SPLINE
SPL {X  -159.701, Y  +348.785, Z    +0.000, E1   +24.361, E3 +434881.176}
SPL {X  -161.904, Y  +363.251, Z    +0.000, E1   +14.606, E3 +434910.971}
SPL {X  -162.745, Y  +375.561, Z    +0.000, E1    +7.538, E3 +434911.168}
SPL {X  -162.820, Y  +385.424, Z    +0.000, E1    +1.080, E3 +434912.062}
SPL {X  -162.820, Y  +389.940, Z    +0.000, E1    -2.281, E3 +434914.938}
SPL {X  -162.820, Y  +396.652, Z    +0.000, E1    -7.520, E3 +434914.517}
SPL {X  -162.820, Y  +406.605, Z    +0.000, E1   -16.760, E3 +434906.994}
SPL {X  -162.820, Y  +420.013, Z    +0.000, E1   -22.833, E3 +434935.115}
SPL {X  -162.820, Y  +442.075, Z    +0.000, E1   -31.090, E3 +434967.901}
ENDSPLINE

SPLINE
SPL {X  -162.820, Y  +436.680, Z    +0.000, E1   -26.151, E3 +434981.205}
ENDSPLINE

SPLINE
SPL {X  -162.820, Y  +438.487, Z    +0.000, E1   -25.409, E3 +434994.844}
SPL {X  -162.820, Y  +441.593, Z    +0.000, E1   -25.391, E3 +435008.452}
SPL {X  -162.820, Y  +444.317, Z    +0.000, E1   -25.492, E3 +435019.634}
SPL {X  -162.820, Y  +446.544, Z    +0.000, E1   -25.427, E3 +435029.803}
SPL {X  -162.820, Y  +448.500, Z    +0.000, E1   -25.425, E3 +435038.405}
SPL {X  -162.820, Y  +451.056, Z    +0.000, E1   -25.443, E3 +435049.512}
SPL {X  -162.820, Y  +454.662, Z    +0.000, E1   -25.474, E3 +435065.256}
SPL {X  -162.820, Y  +458.079, Z    +0.000, E1   -25.369, E3 +435080.835}
SPL {X  -162.820, Y  +460.719, Z    +0.000, E1   -25.411, E3 +435092.094}
SPL {X  -162.820, Y  +463.419, Z    +0.000, E1   -25.510, E3 +435103.131}
SPL {X  -162.820, Y  +465.376, Z    +0.000, E1   -25.372, E3 +435112.719}
SPL {X  -162.820, Y  +467.440, Z    +0.000, E1   -25.427, E3 +435121.351}
SPL {X  -162.820, Y  +470.010, Z    +0.000, E1   -25.445, E3 +435132.555}
SPL {X  -162.820, Y  +473.445, Z    +0.000, E1   -25.493, E3 +435147.279}
SPL {X  -162.820, Y  +476.157, Z    +0.000, E1   -25.426, E3 +435159.494}
SPL {X  -162.820, Y  +478.461, Z    +0.000, E1   -25.410, E3 +435169.774}
SPL {X  -162.820, Y  +481.644, Z    +0.000, E1   -25.433, E3 +435183.720}
SPL {X  -162.820, Y  +486.042, Z    +0.000, E1   -25.483, E3 +435202.639}
SPL {X  -162.820, Y  +490.287, Z    +0.000, E1   -25.463, E3 +435221.358}
SPL {X  -162.820, Y  +494.454, Z    +0.000, E1   -25.465, E3 +435239.589}
SPL {X  -162.820, Y  +498.644, Z    +0.000, E1   -25.463, E3 +435257.965}
SPL {X  -162.820, Y  +502.845, Z    +0.000, E1   -25.458, E3 +435276.399}
SPL {X  -162.820, Y  +506.050, Z    +0.000, E1   -25.420, E3 +435290.538}
SPL {X  -162.820, Y  +508.346, Z    +0.000, E1   -25.444, E3 +435300.387}
SPL {X  -162.820, Y  +511.422, Z    +0.000, E1   -25.445, E3 +435314.047}
SPL {X  -162.820, Y  +515.039, Z    +0.000, E1   -25.452, E3 +435329.728}
SPL {X  -162.820, Y  +517.481, Z    +0.000, E1   -25.432, E3 +435340.463}
SPL {X  -162.820, Y  +519.134, Z    +0.000, E1   -25.366, E3 +435348.210}
SPL {X  -162.820, Y  +521.486, Z    +0.000, E1   -25.382, E3 +435358.506}
SPL {X  -162.820, Y  +525.073, Z    +0.000, E1   -25.512, E3 +435373.312}
SPL {X  -162.820, Y  +527.738, Z    +0.000, E1   -25.438, E3 +435385.360}
SPL {X  -162.820, Y  +530.432, Z    +0.000, E1   -25.477, E3 +435396.937}
SPL {X  -162.820, Y  +534.051, Z    +0.000, E1   -25.484, E3 +435412.814}
SPL {X  -162.820, Y  +537.226, Z    +0.000, E1   -25.378, E3 +435427.383}
SPL {X  -162.820, Y  +539.521, Z    +0.000, E1   -25.386, E3 +435437.342}
SPL {X  -162.820, Y  +542.667, Z    +0.000, E1   -25.474, E3 +435450.667}
SPL {X  -162.820, Y  +546.125, Z    +0.000, E1   -25.505, E3 +435465.392}
SPL {X  -162.820, Y  +548.232, Z    +0.000, E1   -25.424, E3 +435475.154}
SPL {X  -162.820, Y  +550.399, Z    +0.000, E1   -25.424, E3 +435484.705}
SPL {X  -162.820, Y  +553.157, Z    +0.000, E1   -25.443, E3 +435496.679}
SPL {X  -162.820, Y  +556.150, Z    +0.000, E1   -25.445, E3 +435509.769}
SPL {X  -162.820, Y  +559.215, Z    +0.000, E1   -25.460, E3 +435523.071}
SPL {X  -162.820, Y  +562.125, Z    +0.000, E1   -25.434, E3 +435535.991}
SPL {X  -162.820, Y  +564.880, Z    +0.000, E1   -25.448, E3 +435547.945}
SPL {X  -162.820, Y  +568.326, Z    +0.000, E1   -25.470, E3 +435563.005}
SPL {X  -162.820, Y  +572.331, Z    +0.000, E1   -25.489, E3 +435580.380}
SPL {X  -162.820, Y  +576.045, Z    +0.000, E1   -25.412, E3 +435597.188}
SPL {X  -162.820, Y  +580.038, Z    +0.000, E1   -25.473, E3 +435614.283}
SPL {X  -162.820, Y  +583.044, Z    +0.000, E1   -25.450, E3 +435627.406}
SPL {X  -162.820, Y  +585.512, Z    +0.000, E1   -25.448, E3 +435638.302}
SPL {X  -162.820, Y  +588.371, Z    +0.000, E1   -25.460, E3 +435650.688}
SPL {X  -162.820, Y  +590.476, Z    +0.000, E1   -25.398, E3 +435660.329}
SPL {X  -162.820, Y  +593.604, Z    +0.000, E1   -25.477, E3 +435673.607}
SPL {X  -162.820, Y  +596.868, Z    +0.000, E1   -25.461, E3 +435687.873}
SPL {X  -162.820, Y  +599.135, Z    +0.000, E1   -25.398, E3 +435698.242}
SPL {X  -162.820, Y  +601.296, Z    +0.000, E1   -25.399, E3 +435707.723}
SPL {X  -162.820, Y  +603.808, Z    +0.000, E1   -25.554, E3 +435717.511}
SPL {X  -162.820, Y  +607.007, Z    +0.000, E1   -25.491, E3 +435732.202}
SPL {X  -162.820, Y  +611.438, Z    +0.000, E1   -25.467, E3 +435751.792}
SPL {X  -162.820, Y  +615.388, Z    +0.000, E1   -25.455, E3 +435769.051}
SPL {X  -162.820, Y  +618.995, Z    +0.000, E1   -25.483, E3 +435784.646}
SPL {X  -162.820, Y  +622.118, Z    +0.000, E1   -25.492, E3 +435798.111}
SPL {X  -162.820, Y  +624.430, Z    +0.000, E1   -25.475, E3 +435808.332}
SPL {X  -162.820, Y  +626.570, Z    +0.000, E1   -25.441, E3 +435817.932}
SPL {X  -162.820, Y  +628.902, Z    +0.000, E1   -25.449, E3 +435828.113}
SPL {X  -162.820, Y  +631.177, Z    +0.000, E1   -25.467, E3 +435837.944}
SPL {X  -162.820, Y  +633.994, Z    +0.000, E1   -25.503, E3 +435849.990}
SPL {X  -162.820, Y  +636.469, Z    +0.000, E1   -25.465, E3 +435861.034}
SPL {X  -162.820, Y  +638.486, Z    +0.000, E1   -25.456, E3 +435869.952}
SPL {X  -162.820, Y  +640.803, Z    +0.000, E1   -25.462, E3 +435880.013}
SPL {X  -162.820, Y  +643.028, Z    +0.000, E1   -25.494, E3 +435889.522}
SPL {X  -162.820, Y  +645.694, Z    +0.000, E1   -25.540, E3 +435900.810}
SPL {X  -162.820, Y  +649.102, Z    +0.000, E1   -25.495, E3 +435916.238}
SPL {X  -162.820, Y  +652.810, Z    +0.000, E1   -25.497, E3 +435932.272}
SPL {X  -162.820, Y  +655.214, Z    +0.000, E1   -25.485, E3 +435942.774}
SPL {X  -162.820, Y  +657.616, Z    +0.000, E1   -25.511, E3 +435953.129}
SPL {X  -162.820, Y  +660.851, Z    +0.000, E1   -25.520, E3 +435967.271}
SPL {X  -162.820, Y  +663.853, Z    +0.000, E1   -25.496, E3 +435980.453}
SPL {X  -162.820, Y  +667.253, Z    +0.000, E1   -25.483, E3 +435995.625}
SPL {X  -162.820, Y  +671.102, Z    +0.000, E1   -25.514, E3 +436012.076}
SPL {X  -162.820, Y  +673.648, Z    +0.000, E1   -25.431, E3 +436023.742}
SPL {X  -162.796, Y  +676.319, Z    +0.000, E1   -25.526, E3 +436034.752}
SPL {X  -162.707, Y  +679.552, Z    +0.000, E1   -25.443, E3 +436049.626}
SPL {X  -162.545, Y  +682.952, Z    +0.000, E1   -25.510, E3 +436063.859}
SPL {X  -162.381, Y  +685.455, Z    +0.000, E1   -25.410, E3 +436075.546}
SPL {X  -162.194, Y  +687.760, Z    +0.000, E1   -25.360, E3 +436085.982}
SPL {X  -161.866, Y  +691.104, Z    +0.000, E1   -25.383, E3 +436100.614}
SPL {X  -161.319, Y  +695.558, Z    +0.000, E1   -25.832, E3 +436116.416}
SPL {X  -157.976, Y  +712.921, Z    +0.000, E1   -33.197, E3 +436129.808}
ENDSPLINE

SPLINE
SPL {X  -160.738, Y  +699.453, Z    +0.000, E1   -21.994, E3 +436167.435}
SPL {X  -160.945, Y  +698.140, Z    +0.000, E1   -18.412, E3 +436209.674}
SPL {X  -162.497, Y  +683.755, Z    +0.000, E1   -10.754, E3 +436203.818}
SPL {X  -162.819, Y  +673.996, Z    +0.000, E1    -4.745, E3 +436203.419}
ENDSPLINE

SPLINE
SPL {X  -162.791, Y  +676.574, Z    +0.000, E1    -6.127, E3 +436216.107}
ENDSPLINE

SPLINE
SPL {X  -162.820, Y  +667.935, Z    +0.000, E1    -0.509, E3 +436206.193}
SPL {X  -162.820, Y  +662.949, Z    +0.000, E1    +3.113, E3 +436204.312}
SPL {X  -162.820, Y  +658.484, Z    +0.000, E1    +6.336, E3 +436211.457}
SPL {X  -162.820, Y  +640.102, Z    +0.000, E1   +22.409, E3 +436206.196}
SPL {X  -162.820, Y  +633.503, Z    +0.000, E1   +21.975, E3 +436238.433}
SPL {X  -162.820, Y  +611.299, Z    +0.000, E1   +31.088, E3 +436266.545}
ENDSPLINE

SPLINE
SPL {X  -162.820, Y  +618.877, Z    +0.000, E1   +25.259, E3 +436278.040}
ENDSPLINE

SPLINE
SPL {X  -162.820, Y  +617.582, Z    +0.000, E1   +24.552, E3 +436289.416}
SPL {X  -162.820, Y  +614.716, Z    +0.000, E1   +24.535, E3 +436302.628}
SPL {X  -162.820, Y  +611.754, Z    +0.000, E1   +24.563, E3 +436315.916}
SPL {X  -162.820, Y  +608.970, Z    +0.000, E1   +24.542, E3 +436328.756}
SPL {X  -162.820, Y  +606.285, Z    +0.000, E1   +24.533, E3 +436341.092}
SPL {X  -162.820, Y  +603.509, Z    +0.000, E1   +24.546, E3 +436353.629}
SPL {X  -162.820, Y  +600.230, Z    +0.000, E1   +24.589, E3 +436368.374}
SPL {X  -162.820, Y  +597.446, Z    +0.000, E1   +24.542, E3 +436381.232}
SPL {X  -162.820, Y  +595.188, Z    +0.000, E1   +24.538, E3 +436391.623}
SPL {X  -162.820, Y  +592.738, Z    +0.000, E1   +24.551, E3 +436402.671}
SPL {X  -162.820, Y  +590.118, Z    +0.000, E1   +24.544, E3 +436414.731}
SPL {X  -162.820, Y  +587.204, Z    +0.000, E1   +24.592, E3 +436427.607}
SPL {X  -162.820, Y  +584.766, Z    +0.000, E1   +24.499, E3 +436439.441}
SPL {X  -162.820, Y  +581.896, Z    +0.000, E1   +24.528, E3 +436452.383}
SPL {X  -162.820, Y  +579.244, Z    +0.000, E1   +24.610, E3 +436463.727}
SPL {X  -162.820, Y  +576.848, Z    +0.000, E1   +24.543, E3 +436475.268}
SPL {X  -162.820, Y  +573.694, Z    +0.000, E1   +24.535, E3 +436489.738}
SPL {X  -162.820, Y  +571.322, Z    +0.000, E1   +24.492, E3 +436500.771}
SPL {X  -162.820, Y  +568.309, Z    +0.000, E1   +24.589, E3 +436513.996}
SPL {X  -162.820, Y  +564.977, Z    +0.000, E1   +24.571, E3 +436529.169}
SPL {X  -162.820, Y  +562.356, Z    +0.000, E1   +24.575, E3 +436541.068}
SPL {X  -162.820, Y  +558.990, Z    +0.000, E1   +24.558, E3 +436556.718}
SPL {X  -162.820, Y  +555.584, Z    +0.000, E1   +24.559, E3 +436572.087}
SPL {X  -162.820, Y  +552.867, Z    +0.000, E1   +24.583, E3 +436584.282}
SPL {X  -162.820, Y  +549.589, Z    +0.000, E1   +24.547, E3 +436599.648}
SPL {X  -162.820, Y  +546.972, Z    +0.000, E1   +24.516, E3 +436611.613}
SPL {X  -162.820, Y  +544.025, Z    +0.000, E1   +24.611, E3 +436624.558}
SPL {X  -162.820, Y  +540.573, Z    +0.000, E1   +24.503, E3 +436641.012}
SPL {X  -162.820, Y  +538.106, Z    +0.000, E1   +24.553, E3 +436651.766}
SPL {X  -162.820, Y  +536.451, Z    +0.000, E1   +24.519, E3 +436659.584}
SPL {X  -162.820, Y  +534.025, Z    +0.000, E1   +24.589, E3 +436670.184}
SPL {X  -162.820, Y  +531.527, Z    +0.000, E1   +24.582, E3 +436681.570}
SPL {X  -162.820, Y  +529.165, Z    +0.000, E1   +24.521, E3 +436692.819}
SPL {X  -162.820, Y  +525.802, Z    +0.000, E1   +24.585, E3 +436707.839}
SPL {X  -162.820, Y  +521.731, Z    +0.000, E1   +24.542, E3 +436726.775}
SPL {X  -162.820, Y  +518.185, Z    +0.000, E1   +24.561, E3 +436742.647}
SPL {X  -162.820, Y  +508.728, Z    +0.000, E1   +28.484, E3 +436753.187}
SPL {X  -162.820, Y  +500.664, Z    +0.000, E1   +31.476, E3 +436761.851}
SPL {X  -162.820, Y  +499.290, Z    +0.000, E1   +30.657, E3 +436772.133}
SPL {X  -162.820, Y  +497.251, Z    +0.000, E1   +29.634, E3 +436786.608}
SPL {X  -162.820, Y  +495.647, Z    +0.000, E1   +28.606, E3 +436799.485}
SPL {X  -162.820, Y  +494.678, Z    +0.000, E1   +27.647, E3 +436810.186}
SPL {X  -162.820, Y  +493.757, Z    +0.000, E1   +26.462, E3 +436822.546}
SPL {X  -162.820, Y  +492.330, Z    +0.000, E1   +25.953, E3 +436832.300}
SPL {X  -162.820, Y  +489.800, Z    +0.000, E1   +25.653, E3 +436845.761}
SPL {X  -162.820, Y  +485.392, Z    +0.000, E1   +25.667, E3 +436864.789}
SPL {X  -162.820, Y  +482.092, Z    +0.000, E1   +25.593, E3 +436879.477}
SPL {X  -162.820, Y  +479.578, Z    +0.000, E1   +25.634, E3 +436890.120}
SPL {X  -162.820, Y  +477.137, Z    +0.000, E1   +25.632, E3 +436900.699}
SPL {X  -162.820, Y  +473.770, Z    +0.000, E1   +25.664, E3 +436915.245}
SPL {X  -162.820, Y  +469.694, Z    +0.000, E1   +25.657, E3 +436932.976}
SPL {X  -162.820, Y  +465.727, Z    +0.000, E1   +25.676, E3 +436950.019}
SPL {X  -162.820, Y  +463.001, Z    +0.000, E1   +25.614, E3 +436962.135}
SPL {X  -162.820, Y  +459.882, Z    +0.000, E1   +25.674, E3 +436975.435}
SPL {X  -162.820, Y  +456.773, Z    +0.000, E1   +25.591, E3 +436989.382}
SPL {X  -162.820, Y  +454.429, Z    +0.000, E1   +25.642, E3 +436999.149}
SPL {X  -162.820, Y  +451.204, Z    +0.000, E1   +25.672, E3 +437013.176}
SPL {X  -162.820, Y  +447.822, Z    +0.000, E1   +25.664, E3 +437027.660}
SPL {X  -162.820, Y  +445.556, Z    +0.000, E1   +25.626, E3 +437037.791}
SPL {X  -162.820, Y  +442.508, Z    +0.000, E1   +25.657, E3 +437050.885}
SPL {X  -162.820, Y  +439.273, Z    +0.000, E1   +25.576, E3 +437065.522}
SPL {X  -162.820, Y  +436.773, Z    +0.000, E1   +25.602, E3 +437076.087}
SPL {X  -162.820, Y  +433.761, Z    +0.000, E1   +25.681, E3 +437088.766}
SPL {X  -162.820, Y  +430.942, Z    +0.000, E1   +25.597, E3 +437101.451}
SPL {X  -162.820, Y  +428.576, Z    +0.000, E1   +25.647, E3 +437111.389}
SPL {X  -162.820, Y  +426.525, Z    +0.000, E1   +25.610, E3 +437120.496}
SPL {X  -162.820, Y  +423.655, Z    +0.000, E1   +25.628, E3 +437133.056}
SPL {X  -162.820, Y  +419.407, Z    +0.000, E1   +25.665, E3 +437151.248}
SPL {X  -162.820, Y  +415.900, Z    +0.000, E1   +25.638, E3 +437166.517}
SPL {X  -162.820, Y  +413.088, Z    +0.000, E1   +25.644, E3 +437178.674}
SPL {X  -162.820, Y  +410.320, Z    +0.000, E1   +25.604, E3 +437190.992}
SPL {X  -162.820, Y  +407.487, Z    +0.000, E1   +25.617, E3 +437203.200}
SPL {X  -162.820, Y  +405.108, Z    +0.000, E1   +25.535, E3 +437214.168}
SPL {X  -162.820, Y  +401.373, Z    +0.000, E1   +25.736, E3 +437229.004}
SPL {X  -162.820, Y  +398.703, Z    +0.000, E1   +25.586, E3 +437241.501}
SPL {X  -162.820, Y  +395.582, Z    +0.000, E1   +25.684, E3 +437254.493}
SPL {X  -162.820, Y  +391.417, Z    +0.000, E1   +25.659, E3 +437272.831}
SPL {X  -162.820, Y  +387.939, Z    +0.000, E1   +25.627, E3 +437287.978}
SPL {X  -162.820, Y  +385.565, Z    +0.000, E1   +25.686, E3 +437297.766}
SPL {X  -162.820, Y  +383.458, Z    +0.000, E1   +25.657, E3 +437307.130}
SPL {X  -162.820, Y  +381.229, Z    +0.000, E1   +25.660, E3 +437316.806}
SPL {X  -162.797, Y  +377.786, Z    +0.000, E1   +25.638, E3 +437332.095}
SPL {X  -162.663, Y  +373.346, Z    +0.000, E1   +25.707, E3 +437350.834}
SPL {X  -162.487, Y  +370.088, Z    +0.000, E1   +25.525, E3 +437366.169}
SPL {X  -162.307, Y  +367.587, Z    +0.000, E1   +25.577, E3 +437376.587}
SPL {X  -162.041, Y  +364.588, Z    +0.000, E1   +25.591, E3 +437389.665}
SPL {X  -161.695, Y  +361.389, Z    +0.000, E1   +25.445, E3 +437404.551}
SPL {X  -161.190, Y  +357.520, Z    +0.000, E1   +25.774, E3 +437418.802}
SPL {X  -154.424, Y  +328.890, Z    +0.000, E1   +36.591, E3 +437443.802}
ENDSPLINE

SPLINE
SPL {X  -159.701, Y  +348.785, Z    +0.000, E1   +24.361, E3 +437472.085}
SPL {X  -161.904, Y  +363.251, Z    +0.000, E1   +14.606, E3 +437501.880}
SPL {X  -162.745, Y  +375.561, Z    +0.000, E1    +7.538, E3 +437502.077}
SPL {X  -162.820, Y  +385.424, Z    +0.000, E1    +1.080, E3 +437502.971}
SPL {X  -162.820, Y  +389.940, Z    +0.000, E1    -2.281, E3 +437505.847}
SPL {X  -162.820, Y  +396.652, Z    +0.000, E1    -7.520, E3 +437505.426}
SPL {X  -162.820, Y  +406.605, Z    +0.000, E1   -16.760, E3 +437497.903}
SPL {X  -162.820, Y  +418.675, Z    +0.000, E1   -22.201, E3 +437524.151}
SPL {X  -162.820, Y  +425.113, Z    +0.000, E1   -25.243, E3 +437533.088}
SPL {X  -162.820, Y  +442.075, Z    +0.000, E1   -31.090, E3 +437558.810}
ENDSPLINE

SPLINE
SPL {X  -162.820, Y  +436.949, Z    +0.000, E1   -25.871, E3 +437575.560}
ENDSPLINE

SPLINE
SPL {X  -162.820, Y  +439.120, Z    +0.000, E1   -25.352, E3 +437588.809}
SPL {X  -162.820, Y  +441.593, Z    +0.000, E1   -25.391, E3 +437599.361}
SPL {X  -162.820, Y  +444.317, Z    +0.000, E1   -25.492, E3 +437610.543}
SPL {X  -162.820, Y  +447.641, Z    +0.000, E1   -25.460, E3 +437625.478}
SPL {X  -162.820, Y  +451.056, Z    +0.000, E1   -25.443, E3 +437640.421}
SPL {X  -162.820, Y  +454.662, Z    +0.000, E1   -25.474, E3 +437656.165}
SPL {X  -162.820, Y  +458.079, Z    +0.000, E1   -25.369, E3 +437671.745}
SPL {X  -162.820, Y  +460.719, Z    +0.000, E1   -25.411, E3 +437683.003}
SPL {X  -162.820, Y  +463.419, Z    +0.000, E1   -25.510, E3 +437694.040}
SPL {X  -162.820, Y  +465.376, Z    +0.000, E1   -25.372, E3 +437703.628}
SPL {X  -162.820, Y  +467.440, Z    +0.000, E1   -25.427, E3 +437712.260}
SPL {X  -162.820, Y  +470.010, Z    +0.000, E1   -25.445, E3 +437723.464}
SPL {X  -162.820, Y  +473.445, Z    +0.000, E1   -25.493, E3 +437738.188}
SPL {X  -162.820, Y  +476.157, Z    +0.000, E1   -25.426, E3 +437750.403}
SPL {X  -162.820, Y  +478.461, Z    +0.000, E1   -25.410, E3 +437760.683}
SPL {X  -162.820, Y  +481.644, Z    +0.000, E1   -25.433, E3 +437774.629}
SPL {X  -162.820, Y  +486.042, Z    +0.000, E1   -25.483, E3 +437793.548}
SPL {X  -162.820, Y  +490.287, Z    +0.000, E1   -25.463, E3 +437812.267}
SPL {X  -162.820, Y  +494.454, Z    +0.000, E1   -25.465, E3 +437830.498}
SPL {X  -162.820, Y  +498.644, Z    +0.000, E1   -25.463, E3 +437848.874}
SPL {X  -162.820, Y  +502.845, Z    +0.000, E1   -25.458, E3 +437867.308}
SPL {X  -162.820, Y  +506.050, Z    +0.000, E1   -25.420, E3 +437881.447}
SPL {X  -162.820, Y  +508.346, Z    +0.000, E1   -25.444, E3 +437891.296}
SPL {X  -162.820, Y  +511.422, Z    +0.000, E1   -25.445, E3 +437904.956}
SPL {X  -162.820, Y  +515.039, Z    +0.000, E1   -25.452, E3 +437920.638}
SPL {X  -162.820, Y  +517.481, Z    +0.000, E1   -25.432, E3 +437931.372}
SPL {X  -162.820, Y  +519.134, Z    +0.000, E1   -25.366, E3 +437939.119}
SPL {X  -162.820, Y  +521.486, Z    +0.000, E1   -25.382, E3 +437949.415}
SPL {X  -162.820, Y  +525.073, Z    +0.000, E1   -25.512, E3 +437964.221}
SPL {X  -162.820, Y  +527.738, Z    +0.000, E1   -25.438, E3 +437976.269}
SPL {X  -162.820, Y  +530.432, Z    +0.000, E1   -25.477, E3 +437987.846}
SPL {X  -162.820, Y  +534.051, Z    +0.000, E1   -25.484, E3 +438003.723}
SPL {X  -162.820, Y  +537.226, Z    +0.000, E1   -25.378, E3 +438018.292}
SPL {X  -162.820, Y  +539.521, Z    +0.000, E1   -25.386, E3 +438028.251}
SPL {X  -162.820, Y  +542.667, Z    +0.000, E1   -25.474, E3 +438041.576}
SPL {X  -162.820, Y  +546.125, Z    +0.000, E1   -25.505, E3 +438056.301}
SPL {X  -162.820, Y  +549.578, Z    +0.000, E1   -25.462, E3 +438071.925}
SPL {X  -162.820, Y  +553.157, Z    +0.000, E1   -25.443, E3 +438087.588}
SPL {X  -162.820, Y  +556.150, Z    +0.000, E1   -25.445, E3 +438100.678}
SPL {X  -162.820, Y  +559.215, Z    +0.000, E1   -25.460, E3 +438113.980}
SPL {X  -162.820, Y  +562.125, Z    +0.000, E1   -25.434, E3 +438126.900}
SPL {X  -162.820, Y  +564.880, Z    +0.000, E1   -25.448, E3 +438138.854}
SPL {X  -162.820, Y  +568.326, Z    +0.000, E1   -25.470, E3 +438153.914}
SPL {X  -162.820, Y  +572.331, Z    +0.000, E1   -25.489, E3 +438171.289}
SPL {X  -162.820, Y  +576.045, Z    +0.000, E1   -25.412, E3 +438188.097}
SPL {X  -162.820, Y  +580.038, Z    +0.000, E1   -25.473, E3 +438205.192}
SPL {X  -162.820, Y  +583.044, Z    +0.000, E1   -25.450, E3 +438218.315}
SPL {X  -162.820, Y  +585.512, Z    +0.000, E1   -25.448, E3 +438229.211}
SPL {X  -162.820, Y  +588.371, Z    +0.000, E1   -25.460, E3 +438241.597}
SPL {X  -162.820, Y  +590.476, Z    +0.000, E1   -25.398, E3 +438251.238}
SPL {X  -162.820, Y  +593.604, Z    +0.000, E1   -25.477, E3 +438264.516}
SPL {X  -162.820, Y  +596.868, Z    +0.000, E1   -25.461, E3 +438278.782}
SPL {X  -162.820, Y  +599.135, Z    +0.000, E1   -25.398, E3 +438289.151}
SPL {X  -162.820, Y  +601.296, Z    +0.000, E1   -25.399, E3 +438298.632}
SPL {X  -162.820, Y  +603.808, Z    +0.000, E1   -25.554, E3 +438308.420}
SPL {X  -162.820, Y  +607.007, Z    +0.000, E1   -25.491, E3 +438323.111}
SPL {X  -162.820, Y  +611.438, Z    +0.000, E1   -25.467, E3 +438342.701}
SPL {X  -162.820, Y  +615.388, Z    +0.000, E1   -25.455, E3 +438359.960}
SPL {X  -162.820, Y  +618.103, Z    +0.000, E1   -25.456, E3 +438371.708}
SPL {X  -162.820, Y  +621.264, Z    +0.000, E1   -25.514, E3 +438385.310}
SPL {X  -162.820, Y  +624.430, Z    +0.000, E1   -25.475, E3 +438399.241}
SPL {X  -162.820, Y  +626.570, Z    +0.000, E1   -25.441, E3 +438408.842}
SPL {X  -162.820, Y  +628.902, Z    +0.000, E1   -25.449, E3 +438419.022}
SPL {X  -162.820, Y  +631.177, Z    +0.000, E1   -25.467, E3 +438428.853}
SPL {X  -162.820, Y  +633.994, Z    +0.000, E1   -25.503, E3 +438440.899}
SPL {X  -162.820, Y  +637.619, Z    +0.000, E1   -25.497, E3 +438456.959}
SPL {X  -162.820, Y  +640.803, Z    +0.000, E1   -25.462, E3 +438470.922}
SPL {X  -162.820, Y  +643.028, Z    +0.000, E1   -25.494, E3 +438480.432}
SPL {X  -162.820, Y  +646.519, Z    +0.000, E1   -25.551, E3 +438495.414}
SPL {X  -162.820, Y  +649.837, Z    +0.000, E1   -25.446, E3 +438510.538}
SPL {X  -162.820, Y  +652.810, Z    +0.000, E1   -25.497, E3 +438523.181}
SPL {X  -162.820, Y  +655.214, Z    +0.000, E1   -25.485, E3 +438533.683}
SPL {X  -162.820, Y  +657.616, Z    +0.000, E1   -25.511, E3 +438544.038}
SPL {X  -162.820, Y  +660.007, Z    +0.000, E1   -25.550, E3 +438554.099}
SPL {X  -162.820, Y  +662.980, Z    +0.000, E1   -25.505, E3 +438567.657}
SPL {X  -162.820, Y  +667.253, Z    +0.000, E1   -25.483, E3 +438586.534}
SPL {X  -162.820, Y  +671.102, Z    +0.000, E1   -25.514, E3 +438602.985}
SPL {X  -162.820, Y  +673.648, Z    +0.000, E1   -25.431, E3 +438614.651}
SPL {X  -162.796, Y  +676.319, Z    +0.000, E1   -25.526, E3 +438625.661}
SPL {X  -162.739, Y  +678.625, Z    +0.000, E1   -25.423, E3 +438636.452}
SPL {X  -162.669, Y  +680.515, Z    +0.000, E1   -25.398, E3 +438644.907}
SPL {X  -162.545, Y  +682.952, Z    +0.000, E1   -25.510, E3 +438654.768}
SPL {X  -162.381, Y  +685.455, Z    +0.000, E1   -25.410, E3 +438666.455}
SPL {X  -162.194, Y  +687.760, Z    +0.000, E1   -25.360, E3 +438676.891}
SPL {X  -161.866, Y  +691.104, Z    +0.000, E1   -25.383, E3 +438691.523}
SPL {X  -161.319, Y  +695.558, Z    +0.000, E1   -25.832, E3 +438707.325}
SPL {X  -157.976, Y  +712.921, Z    +0.000, E1   -33.197, E3 +438720.717}
ENDSPLINE

SPLINE
SPL {X  -160.738, Y  +699.453, Z    +0.000, E1   -21.994, E3 +438758.344}
SPL {X  -160.945, Y  +698.140, Z    +0.000, E1   -18.412, E3 +438800.584}
SPL {X  -162.497, Y  +683.755, Z    +0.000, E1   -10.754, E3 +438794.727}
SPL {X  -162.819, Y  +673.996, Z    +0.000, E1    -4.745, E3 +438794.328}
ENDSPLINE

SPLINE
SPL {X  -162.791, Y  +676.574, Z    +0.000, E1    -6.127, E3 +438807.016}
ENDSPLINE

SPLINE
SPL {X  -162.820, Y  +667.935, Z    +0.000, E1    -0.509, E3 +438797.102}
SPL {X  -162.820, Y  +662.949, Z    +0.000, E1    +3.113, E3 +438795.221}
SPL {X  -162.820, Y  +658.484, Z    +0.000, E1    +6.336, E3 +438802.367}
SPL {X  -162.820, Y  +640.102, Z    +0.000, E1   +22.409, E3 +438797.105}
SPL {X  -162.820, Y  +633.503, Z    +0.000, E1   +21.975, E3 +438829.342}
SPL {X  -162.820, Y  +611.299, Z    +0.000, E1   +31.088, E3 +438857.454}
ENDSPLINE

SPLINE
SPL {X  -162.820, Y  +618.877, Z    +0.000, E1   +25.259, E3 +438868.949}
ENDSPLINE

SPLINE
SPL {X  -162.820, Y  +617.582, Z    +0.000, E1   +24.552, E3 +438880.325}
SPL {X  -162.820, Y  +614.716, Z    +0.000, E1   +24.535, E3 +438893.537}
SPL {X  -162.820, Y  +611.754, Z    +0.000, E1   +24.563, E3 +438906.825}
SPL {X  -162.820, Y  +608.970, Z    +0.000, E1   +24.542, E3 +438919.665}
SPL {X  -162.820, Y  +606.285, Z    +0.000, E1   +24.533, E3 +438932.001}
SPL {X  -162.820, Y  +603.509, Z    +0.000, E1   +24.546, E3 +438944.538}
SPL {X  -162.820, Y  +600.818, Z    +0.000, E1   +24.590, E3 +438956.461}
SPL {X  -162.820, Y  +598.053, Z    +0.000, E1   +24.547, E3 +438969.444}
SPL {X  -162.820, Y  +595.188, Z    +0.000, E1   +24.538, E3 +438982.532}
SPL {X  -162.820, Y  +592.738, Z    +0.000, E1   +24.551, E3 +438993.580}
SPL {X  -162.820, Y  +590.118, Z    +0.000, E1   +24.544, E3 +439005.640}
SPL {X  -162.820, Y  +587.204, Z    +0.000, E1   +24.592, E3 +439018.517}
SPL {X  -162.820, Y  +584.193, Z    +0.000, E1   +24.484, E3 +439033.227}
SPL {X  -162.820, Y  +581.176, Z    +0.000, E1   +24.592, E3 +439045.988}
SPL {X  -162.820, Y  +578.588, Z    +0.000, E1   +24.598, E3 +439057.843}
SPL {X  -162.820, Y  +576.196, Z    +0.000, E1   +24.519, E3 +439069.227}
SPL {X  -162.820, Y  +573.694, Z    +0.000, E1   +24.535, E3 +439080.647}
SPL {X  -162.820, Y  +570.310, Z    +0.000, E1   +24.556, E3 +439095.963}
SPL {X  -162.820, Y  +567.494, Z    +0.000, E1   +24.547, E3 +439108.748}
SPL {X  -162.820, Y  +564.977, Z    +0.000, E1   +24.571, E3 +439120.078}
SPL {X  -162.820, Y  +562.356, Z    +0.000, E1   +24.575, E3 +439131.977}
SPL {X  -162.820, Y  +558.990, Z    +0.000, E1   +24.558, E3 +439147.627}
SPL {X  -162.820, Y  +555.584, Z    +0.000, E1   +24.559, E3 +439162.996}
SPL {X  -162.820, Y  +552.867, Z    +0.000, E1   +24.583, E3 +439175.191}
SPL {X  -162.820, Y  +549.589, Z    +0.000, E1   +24.547, E3 +439190.557}
SPL {X  -162.820, Y  +545.742, Z    +0.000, E1   +24.577, E3 +439207.844}
SPL {X  -162.820, Y  +542.970, Z    +0.000, E1   +24.579, E3 +439220.287}
SPL {X  -162.820, Y  +540.573, Z    +0.000, E1   +24.503, E3 +439231.921}
SPL {X  -162.820, Y  +538.106, Z    +0.000, E1   +24.553, E3 +439242.675}
SPL {X  -162.820, Y  +536.451, Z    +0.000, E1   +24.519, E3 +439250.493}
SPL {X  -162.820, Y  +534.025, Z    +0.000, E1   +24.589, E3 +439261.093}
SPL {X  -162.820, Y  +531.527, Z    +0.000, E1   +24.582, E3 +439272.479}
SPL {X  -162.820, Y  +529.165, Z    +0.000, E1   +24.521, E3 +439283.728}
SPL {X  -162.820, Y  +525.802, Z    +0.000, E1   +24.585, E3 +439298.748}
SPL {X  -162.820, Y  +521.731, Z    +0.000, E1   +24.542, E3 +439317.684}
SPL {X  -162.820, Y  +518.185, Z    +0.000, E1   +24.561, E3 +439333.556}
SPL {X  -162.820, Y  +508.728, Z    +0.000, E1   +28.484, E3 +439344.096}
SPL {X  -162.820, Y  +500.664, Z    +0.000, E1   +31.476, E3 +439352.760}
SPL {X  -162.820, Y  +499.290, Z    +0.000, E1   +30.657, E3 +439363.042}
SPL {X  -162.820, Y  +497.251, Z    +0.000, E1   +29.634, E3 +439377.518}
SPL {X  -162.820, Y  +495.647, Z    +0.000, E1   +28.606, E3 +439390.394}
SPL {X  -162.820, Y  +494.678, Z    +0.000, E1   +27.647, E3 +439401.095}
SPL {X  -162.820, Y  +493.757, Z    +0.000, E1   +26.462, E3 +439413.455}
SPL {X  -162.820, Y  +492.330, Z    +0.000, E1   +25.953, E3 +439423.209}
SPL {X  -162.820, Y  +490.849, Z    +0.000, E1   +25.593, E3 +439432.372}
SPL {X  -162.820, Y  +487.351, Z    +0.000, E1   +25.663, E3 +439447.232}
SPL {X  -162.820, Y  +484.247, Z    +0.000, E1   +25.651, E3 +439460.559}
SPL {X  -162.820, Y  +482.092, Z    +0.000, E1   +25.593, E3 +439470.386}
SPL {X  -162.820, Y  +479.578, Z    +0.000, E1   +25.634, E3 +439481.029}
SPL {X  -162.820, Y  +477.137, Z    +0.000, E1   +25.632, E3 +439491.608}
SPL {X  -162.820, Y  +473.770, Z    +0.000, E1   +25.664, E3 +439506.154}
SPL {X  -162.820, Y  +470.744, Z    +0.000, E1   +25.641, E3 +439519.251}
SPL {X  -162.820, Y  +467.745, Z    +0.000, E1   +25.668, E3 +439532.233}
SPL {X  -162.820, Y  +463.978, Z    +0.000, E1   +25.651, E3 +439548.710}
SPL {X  -162.820, Y  +460.810, Z    +0.000, E1   +25.619, E3 +439562.568}
SPL {X  -162.820, Y  +457.479, Z    +0.000, E1   +25.656, E3 +439576.914}
SPL {X  -162.820, Y  +453.678, Z    +0.000, E1   +25.652, E3 +439593.366}
SPL {X  -162.820, Y  +450.466, Z    +0.000, E1   +25.644, E3 +439607.311}
SPL {X  -162.820, Y  +447.822, Z    +0.000, E1   +25.664, E3 +439618.569}
SPL {X  -162.820, Y  +444.499, Z    +0.000, E1   +25.673, E3 +439633.139}
SPL {X  -162.820, Y  +440.857, Z    +0.000, E1   +25.614, E3 +439649.248}
SPL {X  -162.820, Y  +438.582, Z    +0.000, E1   +25.544, E3 +439659.568}
SPL {X  -162.820, Y  +435.635, Z    +0.000, E1   +25.661, E3 +439671.663}
SPL {X  -162.820, Y  +432.815, Z    +0.000, E1   +25.641, E3 +439683.892}
SPL {X  -162.820, Y  +430.942, Z    +0.000, E1   +25.597, E3 +439692.360}
SPL {X  -162.820, Y  +428.576, Z    +0.000, E1   +25.647, E3 +439702.298}
SPL {X  -162.820, Y  +426.525, Z    +0.000, E1   +25.610, E3 +439711.405}
SPL {X  -162.820, Y  +423.655, Z    +0.000, E1   +25.628, E3 +439723.965}
SPL {X  -162.820, Y  +419.407, Z    +0.000, E1   +25.665, E3 +439742.157}
SPL {X  -162.820, Y  +415.900, Z    +0.000, E1   +25.638, E3 +439757.426}
SPL {X  -162.820, Y  +413.088, Z    +0.000, E1   +25.644, E3 +439769.583}
SPL {X  -162.820, Y  +410.320, Z    +0.000, E1   +25.604, E3 +439781.901}
SPL {X  -162.820, Y  +407.487, Z    +0.000, E1   +25.617, E3 +439794.109}
SPL {X  -162.820, Y  +405.108, Z    +0.000, E1   +25.535, E3 +439805.077}
SPL {X  -162.820, Y  +401.373, Z    +0.000, E1   +25.736, E3 +439819.913}
SPL {X  -162.820, Y  +398.703, Z    +0.000, E1   +25.586, E3 +439832.410}
SPL {X  -162.820, Y  +395.582, Z    +0.000, E1   +25.684, E3 +439845.402}
SPL {X  -162.820, Y  +391.417, Z    +0.000, E1   +25.659, E3 +439863.740}
SPL {X  -162.820, Y  +387.939, Z    +0.000, E1   +25.627, E3 +439878.887}
SPL {X  -162.820, Y  +385.565, Z    +0.000, E1   +25.686, E3 +439888.676}
SPL {X  -162.820, Y  +383.458, Z    +0.000, E1   +25.657, E3 +439898.040}
SPL {X  -162.820, Y  +380.448, Z    +0.000, E1   +25.674, E3 +439911.148}
SPL {X  -162.785, Y  +377.106, Z    +0.000, E1   +25.598, E3 +439926.092}
SPL {X  -162.709, Y  +374.484, Z    +0.000, E1   +25.711, E3 +439936.543}
SPL {X  -162.623, Y  +372.485, Z    +0.000, E1   +25.631, E3 +439945.824}
SPL {X  -162.487, Y  +370.088, Z    +0.000, E1   +25.525, E3 +439957.078}
SPL {X  -162.243, Y  +366.801, Z    +0.000, E1   +25.618, E3 +439970.718}
SPL {X  -161.977, Y  +363.953, Z    +0.000, E1   +25.528, E3 +439983.645}
SPL {X  -161.695, Y  +361.389, Z    +0.000, E1   +25.445, E3 +439995.460}
SPL {X  -161.364, Y  +358.774, Z    +0.000, E1   +25.454, E3 +440006.660}
SPL {X  -160.939, Y  +355.820, Z    +0.000, E1   +26.179, E3 +440013.879}
SPL {X  -155.035, Y  +330.756, Z    +0.000, E1   +37.918, E3 +440020.212}
SPL {X  -153.918, Y  +327.401, Z    +0.000, E1   +34.677, E3 +440055.513}
ENDSPLINE

SPLINE
SPL {X  -159.701, Y  +348.785, Z    +0.000, E1   +24.361, E3 +440062.994}
SPL {X  -162.442, Y  +369.407, Z    +0.000, E1   +11.234, E3 +440092.629}
SPL {X  -162.820, Y  +384.333, Z    +0.000, E1    +1.902, E3 +440093.835}
SPL {X  -162.820, Y  +389.940, Z    +0.000, E1    -2.281, E3 +440096.756}
SPL {X  -162.820, Y  +396.652, Z    +0.000, E1    -7.520, E3 +440096.335}
SPL {X  -162.820, Y  +409.181, Z    +0.000, E1   -18.650, E3 +440090.554}
SPL {X  -162.820, Y  +419.618, Z    +0.000, E1   -22.332, E3 +440118.036}
SPL {X  -162.820, Y  +442.075, Z    +0.000, E1   -31.090, E3 +440149.719}
ENDSPLINE

SPLINE
SPL {X  -162.820, Y  +436.949, Z    +0.000, E1   -25.871, E3 +440166.469}
ENDSPLINE

SPLINE
SPL {X  -162.820, Y  +439.120, Z    +0.000, E1   -25.352, E3 +440179.719}
SPL {X  -162.820, Y  +441.593, Z    +0.000, E1   -25.391, E3 +440190.270}
SPL {X  -162.820, Y  +444.317, Z    +0.000, E1   -25.492, E3 +440201.452}
SPL {X  -162.820, Y  +447.641, Z    +0.000, E1   -25.460, E3 +440216.387}
SPL {X  -162.820, Y  +451.939, Z    +0.000, E1   -25.468, E3 +440235.207}
SPL {X  -162.820, Y  +455.480, Z    +0.000, E1   -25.454, E3 +440250.618}
SPL {X  -162.820, Y  +458.079, Z    +0.000, E1   -25.369, E3 +440262.654}
SPL {X  -162.820, Y  +460.719, Z    +0.000, E1   -25.411, E3 +440273.912}
SPL {X  -162.820, Y  +463.419, Z    +0.000, E1   -25.510, E3 +440284.949}
SPL {X  -162.820, Y  +465.376, Z    +0.000, E1   -25.372, E3 +440294.537}
SPL {X  -162.820, Y  +467.440, Z    +0.000, E1   -25.427, E3 +440303.169}
SPL {X  -162.820, Y  +470.010, Z    +0.000, E1   -25.445, E3 +440314.373}
SPL {X  -162.820, Y  +473.445, Z    +0.000, E1   -25.493, E3 +440329.097}
SPL {X  -162.820, Y  +476.157, Z    +0.000, E1   -25.426, E3 +440341.312}
SPL {X  -162.820, Y  +478.461, Z    +0.000, E1   -25.410, E3 +440351.592}
SPL {X  -162.820, Y  +481.644, Z    +0.000, E1   -25.433, E3 +440365.538}
SPL {X  -162.820, Y  +486.042, Z    +0.000, E1   -25.483, E3 +440384.458}
SPL {X  -162.820, Y  +490.287, Z    +0.000, E1   -25.463, E3 +440403.176}
SPL {X  -162.820, Y  +494.454, Z    +0.000, E1   -25.465, E3 +440421.407}
SPL {X  -162.820, Y  +498.644, Z    +0.000, E1   -25.463, E3 +440439.784}
SPL {X  -162.820, Y  +502.845, Z    +0.000, E1   -25.458, E3 +440458.217}
SPL {X  -162.820, Y  +506.050, Z    +0.000, E1   -25.420, E3 +440472.357}
SPL {X  -162.820, Y  +508.346, Z    +0.000, E1   -25.444, E3 +440482.205}
SPL {X  -162.820, Y  +510.377, Z    +0.000, E1   -25.398, E3 +440491.451}
SPL {X  -162.820, Y  +513.176, Z    +0.000, E1   -25.443, E3 +440503.495}
SPL {X  -162.820, Y  +516.690, Z    +0.000, E1   -25.465, E3 +440518.706}
SPL {X  -162.820, Y  +519.134, Z    +0.000, E1   -25.366, E3 +440530.028}
SPL {X  -162.820, Y  +521.486, Z    +0.000, E1   -25.382, E3 +440540.324}
SPL {X  -162.820, Y  +525.073, Z    +0.000, E1   -25.512, E3 +440555.130}
SPL {X  -162.820, Y  +527.738, Z    +0.000, E1   -25.438, E3 +440567.178}
SPL {X  -162.820, Y  +530.432, Z    +0.000, E1   -25.477, E3 +440578.755}
SPL {X  -162.820, Y  +534.051, Z    +0.000, E1   -25.484, E3 +440594.632}
SPL {X  -162.820, Y  +537.226, Z    +0.000, E1   -25.378, E3 +440609.201}
SPL {X  -162.820, Y  +539.521, Z    +0.000, E1   -25.386, E3 +440619.160}
SPL {X  -162.820, Y  +542.667, Z    +0.000, E1   -25.474, E3 +440632.485}
SPL {X  -162.820, Y  +546.125, Z    +0.000, E1   -25.505, E3 +440647.210}
SPL {X  -162.820, Y  +548.232, Z    +0.000, E1   -25.424, E3 +440656.972}
SPL {X  -162.820, Y  +550.399, Z    +0.000, E1   -25.424, E3 +440666.523}
SPL {X  -162.820, Y  +553.157, Z    +0.000, E1   -25.443, E3 +440678.497}
SPL {X  -162.820, Y  +556.150, Z    +0.000, E1   -25.445, E3 +440691.587}
SPL {X  -162.820, Y  +559.215, Z    +0.000, E1   -25.460, E3 +440704.889}
SPL {X  -162.820, Y  +562.125, Z    +0.000, E1   -25.434, E3 +440717.809}
SPL {X  -162.820, Y  +564.880, Z    +0.000, E1   -25.448, E3 +440729.763}
SPL {X  -162.820, Y  +568.326, Z    +0.000, E1   -25.470, E3 +440744.823}
SPL {X  -162.820, Y  +571.303, Z    +0.000, E1   -25.427, E3 +440757.995}
SPL {X  -162.820, Y  +574.067, Z    +0.000, E1   -25.459, E3 +440769.935}
SPL {X  -162.820, Y  +576.597, Z    +0.000, E1   -25.400, E3 +440781.406}
SPL {X  -162.820, Y  +578.977, Z    +0.000, E1   -25.460, E3 +440791.338}
SPL {X  -162.820, Y  +581.995, Z    +0.000, E1   -25.468, E3 +440804.696}
SPL {X  -162.820, Y  +585.512, Z    +0.000, E1   -25.448, E3 +440820.120}
SPL {X  -162.820, Y  +588.371, Z    +0.000, E1   -25.460, E3 +440832.506}
SPL {X  -162.820, Y  +590.476, Z    +0.000, E1   -25.398, E3 +440842.147}
SPL {X  -162.820, Y  +593.604, Z    +0.000, E1   -25.477, E3 +440855.426}
SPL {X  -162.820, Y  +596.868, Z    +0.000, E1   -25.461, E3 +440869.691}
SPL {X  -162.820, Y  +599.135, Z    +0.000, E1   -25.398, E3 +440880.060}
SPL {X  -162.820, Y  +601.296, Z    +0.000, E1   -25.399, E3 +440889.542}
SPL {X  -162.820, Y  +603.808, Z    +0.000, E1   -25.554, E3 +440899.330}
SPL {X  -162.820, Y  +607.007, Z    +0.000, E1   -25.491, E3 +440914.021}
SPL {X  -162.820, Y  +611.438, Z    +0.000, E1   -25.467, E3 +440933.610}
SPL {X  -162.820, Y  +615.388, Z    +0.000, E1   -25.455, E3 +440950.869}
SPL {X  -162.820, Y  +618.995, Z    +0.000, E1   -25.483, E3 +440966.464}
SPL {X  -162.820, Y  +622.118, Z    +0.000, E1   -25.492, E3 +440979.929}
SPL {X  -162.820, Y  +624.430, Z    +0.000, E1   -25.475, E3 +440990.150}
SPL {X  -162.820, Y  +626.570, Z    +0.000, E1   -25.441, E3 +440999.751}
SPL {X  -162.820, Y  +628.902, Z    +0.000, E1   -25.449, E3 +441009.931}
SPL {X  -162.820, Y  +631.177, Z    +0.000, E1   -25.467, E3 +441019.762}
SPL {X  -162.820, Y  +633.994, Z    +0.000, E1   -25.503, E3 +441031.809}
SPL {X  -162.820, Y  +637.619, Z    +0.000, E1   -25.497, E3 +441047.868}
SPL {X  -162.820, Y  +640.803, Z    +0.000, E1   -25.462, E3 +441061.831}
SPL {X  -162.820, Y  +643.028, Z    +0.000, E1   -25.494, E3 +441071.341}
SPL {X  -162.820, Y  +646.519, Z    +0.000, E1   -25.551, E3 +441086.323}
SPL {X  -162.820, Y  +649.837, Z    +0.000, E1   -25.446, E3 +441101.447}
SPL {X  -162.820, Y  +652.810, Z    +0.000, E1   -25.497, E3 +441114.090}
SPL {X  -162.820, Y  +655.214, Z    +0.000, E1   -25.485, E3 +441124.593}
SPL {X  -162.820, Y  +657.616, Z    +0.000, E1   -25.511, E3 +441134.947}
SPL {X  -162.820, Y  +660.851, Z    +0.000, E1   -25.520, E3 +441149.090}
SPL {X  -162.820, Y  +663.853, Z    +0.000, E1   -25.496, E3 +441162.271}
SPL {X  -162.820, Y  +666.096, Z    +0.000, E1   -25.408, E3 +441172.738}
SPL {X  -162.820, Y  +669.195, Z    +0.000, E1   -25.525, E3 +441185.575}
SPL {X  -162.820, Y  +672.979, Z    +0.000, E1   -25.478, E3 +441202.425}
SPL {X  -162.796, Y  +676.319, Z    +0.000, E1   -25.526, E3 +441216.570}
SPL {X  -162.739, Y  +678.625, Z    +0.000, E1   -25.423, E3 +441227.361}
SPL {X  -162.669, Y  +680.515, Z    +0.000, E1   -25.398, E3 +441235.816}
SPL {X  -162.545, Y  +682.952, Z    +0.000, E1   -25.510, E3 +441245.678}
SPL {X  -162.381, Y  +685.455, Z    +0.000, E1   -25.410, E3 +441257.364}
SPL {X  -162.194, Y  +687.760, Z    +0.000, E1   -25.360, E3 +441267.800}
SPL {X  -161.987, Y  +689.945, Z    +0.000, E1   -25.406, E3 +441276.953}
SPL {X  -161.711, Y  +692.468, Z    +0.000, E1   -25.300, E3 +441288.951}
SPL {X  -161.141, Y  +696.825, Z    +0.000, E1   -26.170, E3 +441301.085}
SPL {X  -157.976, Y  +712.921, Z    +0.000, E1   -33.197, E3 +441311.626}
ENDSPLINE

SPLINE
SPL {X  -160.738, Y  +699.453, Z    +0.000, E1   -21.994, E3 +441349.253}
SPL {X  -161.689, Y  +692.657, Z    +0.000, E1   -15.656, E3 +441389.323}
SPL {X  -162.807, Y  +675.545, Z    +0.000, E1    -5.787, E3 +441384.822}
ENDSPLINE

SPLINE
SPL {X  -162.791, Y  +676.574, Z    +0.000, E1    -6.127, E3 +441397.925}
ENDSPLINE

SPLINE
SPL {X  -162.820, Y  +666.063, Z    +0.000, E1    +0.780, E3 +441386.019}
SPL {X  -162.820, Y  +659.251, Z    +0.000, E1    +5.716, E3 +441392.235}
SPL {X  -162.820, Y  +640.102, Z    +0.000, E1   +22.409, E3 +441388.014}
SPL {X  -162.820, Y  +633.503, Z    +0.000, E1   +21.975, E3 +441420.251}
SPL {X  -162.820, Y  +611.299, Z    +0.000, E1   +31.088, E3 +441448.363}
ENDSPLINE

SPLINE
SPL {X  -162.820, Y  +618.877, Z    +0.000, E1   +25.259, E3 +441459.858}
ENDSPLINE

SPLINE
SPL {X  -162.820, Y  +617.582, Z    +0.000, E1   +24.552, E3 +441471.235}
SPL {X  -162.820, Y  +614.716, Z    +0.000, E1   +24.535, E3 +441484.446}
SPL {X  -162.820, Y  +611.754, Z    +0.000, E1   +24.563, E3 +441497.734}
SPL {X  -162.820, Y  +608.970, Z    +0.000, E1   +24.542, E3 +441510.574}
SPL {X  -162.820, Y  +606.285, Z    +0.000, E1   +24.533, E3 +441522.910}
SPL {X  -162.820, Y  +603.509, Z    +0.000, E1   +24.546, E3 +441535.447}
SPL {X  -162.820, Y  +600.818, Z    +0.000, E1   +24.590, E3 +441547.370}
SPL {X  -162.820, Y  +598.053, Z    +0.000, E1   +24.547, E3 +441560.353}
SPL {X  -162.820, Y  +595.188, Z    +0.000, E1   +24.538, E3 +441573.441}
SPL {X  -162.820, Y  +592.738, Z    +0.000, E1   +24.551, E3 +441584.490}
SPL {X  -162.820, Y  +590.118, Z    +0.000, E1   +24.544, E3 +441596.549}
SPL {X  -162.820, Y  +587.204, Z    +0.000, E1   +24.592, E3 +441609.426}
SPL {X  -162.820, Y  +584.766, Z    +0.000, E1   +24.499, E3 +441621.259}
SPL {X  -162.820, Y  +581.896, Z    +0.000, E1   +24.528, E3 +441634.201}
SPL {X  -162.820, Y  +579.244, Z    +0.000, E1   +24.610, E3 +441645.545}
SPL {X  -162.820, Y  +576.848, Z    +0.000, E1   +24.543, E3 +441657.086}
SPL {X  -162.820, Y  +574.433, Z    +0.000, E1   +24.551, E3 +441667.917}
SPL {X  -162.820, Y  +572.074, Z    +0.000, E1   +24.505, E3 +441679.188}
SPL {X  -162.820, Y  +568.309, Z    +0.000, E1   +24.589, E3 +441695.815}
SPL {X  -162.820, Y  +564.977, Z    +0.000, E1   +24.571, E3 +441710.987}
SPL {X  -162.820, Y  +562.356, Z    +0.000, E1   +24.575, E3 +441722.886}
SPL {X  -162.820, Y  +558.990, Z    +0.000, E1   +24.558, E3 +441738.536}
SPL {X  -162.820, Y  +555.584, Z    +0.000, E1   +24.559, E3 +441753.905}
SPL {X  -162.820, Y  +552.169, Z    +0.000, E1   +24.581, E3 +441769.474}
SPL {X  -162.820, Y  +548.172, Z    +0.000, E1   +24.564, E3 +441787.822}
SPL {X  -162.820, Y  +544.025, Z    +0.000, E1   +24.611, E3 +441806.376}
SPL {X  -162.820, Y  +540.573, Z    +0.000, E1   +24.503, E3 +441822.830}
SPL {X  -162.820, Y  +537.211, Z    +0.000, E1   +24.561, E3 +441837.759}
SPL {X  -162.820, Y  +534.025, Z    +0.000, E1   +24.589, E3 +441852.003}
SPL {X  -162.820, Y  +531.527, Z    +0.000, E1   +24.582, E3 +441863.388}
SPL {X  -162.820, Y  +529.165, Z    +0.000, E1   +24.521, E3 +441874.637}
SPL {X  -162.820, Y  +526.822, Z    +0.000, E1   +24.559, E3 +441885.000}
SPL {X  -162.820, Y  +524.112, Z    +0.000, E1   +24.542, E3 +441897.617}
SPL {X  -162.820, Y  +521.048, Z    +0.000, E1   +24.515, E3 +441911.754}
SPL {X  -162.820, Y  +518.185, Z    +0.000, E1   +24.561, E3 +441924.465}
SPL {X  -162.820, Y  +508.728, Z    +0.000, E1   +28.484, E3 +441935.005}
SPL {X  -162.820, Y  +500.664, Z    +0.000, E1   +31.476, E3 +441943.669}
SPL {X  -162.820, Y  +499.290, Z    +0.000, E1   +30.657, E3 +441953.951}
SPL {X  -162.820, Y  +497.700, Z    +0.000, E1   +29.785, E3 +441965.566}
SPL {X  -162.820, Y  +495.915, Z    +0.000, E1   +28.861, E3 +441978.658}
SPL {X  -162.820, Y  +494.678, Z    +0.000, E1   +27.647, E3 +441992.004}
SPL {X  -162.820, Y  +493.757, Z    +0.000, E1   +26.462, E3 +442004.364}
SPL {X  -162.820, Y  +491.420, Z    +0.000, E1   +25.780, E3 +442019.625}
SPL {X  -162.820, Y  +487.351, Z    +0.000, E1   +25.663, E3 +442038.142}
SPL {X  -162.820, Y  +484.247, Z    +0.000, E1   +25.651, E3 +442051.468}
SPL {X  -162.820, Y  +482.092, Z    +0.000, E1   +25.593, E3 +442061.295}
SPL {X  -162.820, Y  +479.578, Z    +0.000, E1   +25.634, E3 +442071.938}
SPL {X  -162.820, Y  +477.137, Z    +0.000, E1   +25.632, E3 +442082.517}
SPL {X  -162.820, Y  +473.770, Z    +0.000, E1   +25.664, E3 +442097.063}
SPL {X  -162.820, Y  +469.694, Z    +0.000, E1   +25.657, E3 +442114.794}
SPL {X  -162.820, Y  +465.727, Z    +0.000, E1   +25.676, E3 +442131.837}
SPL {X  -162.820, Y  +463.001, Z    +0.000, E1   +25.614, E3 +442143.953}
SPL {X  -162.820, Y  +459.882, Z    +0.000, E1   +25.674, E3 +442157.254}
SPL {X  -162.820, Y  +456.773, Z    +0.000, E1   +25.591, E3 +442171.200}
SPL {X  -162.820, Y  +454.429, Z    +0.000, E1   +25.642, E3 +442180.968}
SPL {X  -162.820, Y  +451.204, Z    +0.000, E1   +25.672, E3 +442194.994}
SPL {X  -162.820, Y  +447.822, Z    +0.000, E1   +25.664, E3 +442209.478}
SPL {X  -162.820, Y  +445.556, Z    +0.000, E1   +25.626, E3 +442219.609}
SPL {X  -162.820, Y  +442.508, Z    +0.000, E1   +25.657, E3 +442232.703}
SPL {X  -162.820, Y  +439.273, Z    +0.000, E1   +25.576, E3 +442247.341}
SPL {X  -162.820, Y  +436.773, Z    +0.000, E1   +25.602, E3 +442257.905}
SPL {X  -162.820, Y  +433.761, Z    +0.000, E1   +25.681, E3 +442270.584}
SPL {X  -162.820, Y  +430.942, Z    +0.000, E1   +25.597, E3 +442283.269}
SPL {X  -162.820, Y  +428.576, Z    +0.000, E1   +25.647, E3 +442293.207}
SPL {X  -162.820, Y  +426.525, Z    +0.000, E1   +25.610, E3 +442302.314}
SPL {X  -162.820, Y  +423.655, Z    +0.000, E1   +25.628, E3 +442314.874}
SPL {X  -162.820, Y  +419.407, Z    +0.000, E1   +25.665, E3 +442333.066}
SPL {X  -162.820, Y  +415.900, Z    +0.000, E1   +25.638, E3 +442348.335}
SPL {X  -162.820, Y  +413.088, Z    +0.000, E1   +25.644, E3 +442360.492}
SPL {X  -162.820, Y  +410.320, Z    +0.000, E1   +25.604, E3 +442372.810}
SPL {X  -162.820, Y  +407.487, Z    +0.000, E1   +25.617, E3 +442385.018}
SPL {X  -162.820, Y  +405.108, Z    +0.000, E1   +25.535, E3 +442395.986}
SPL {X  -162.820, Y  +401.373, Z    +0.000, E1   +25.736, E3 +442410.822}
SPL {X  -162.820, Y  +397.357, Z    +0.000, E1   +25.652, E3 +442428.893}
SPL {X  -162.820, Y  +393.659, Z    +0.000, E1   +25.666, E3 +442444.693}
SPL {X  -162.820, Y  +390.679, Z    +0.000, E1   +25.624, E3 +442457.936}
SPL {X  -162.820, Y  +387.939, Z    +0.000, E1   +25.627, E3 +442469.796}
SPL {X  -162.820, Y  +384.398, Z    +0.000, E1   +25.707, E3 +442484.694}
SPL {X  -162.820, Y  +380.448, Z    +0.000, E1   +25.674, E3 +442502.057}
SPL {X  -162.785, Y  +377.106, Z    +0.000, E1   +25.598, E3 +442517.001}
SPL {X  -162.709, Y  +374.484, Z    +0.000, E1   +25.711, E3 +442527.452}
SPL {X  -162.623, Y  +372.485, Z    +0.000, E1   +25.631, E3 +442536.733}
SPL {X  -162.487, Y  +370.088, Z    +0.000, E1   +25.525, E3 +442547.987}
SPL {X  -162.243, Y  +366.801, Z    +0.000, E1   +25.618, E3 +442561.627}
SPL {X  -161.882, Y  +363.046, Z    +0.000, E1   +25.550, E3 +442578.511}
SPL {X  -161.454, Y  +359.455, Z    +0.000, E1   +25.428, E3 +442594.905}
SPL {X  -160.939, Y  +355.820, Z    +0.000, E1   +26.179, E3 +442604.788}
SPL {X  -154.424, Y  +328.890, Z    +0.000, E1   +36.591, E3 +442625.620}
ENDSPLINE

SPLINE
SPL {X  -159.701, Y  +348.785, Z    +0.000, E1   +24.361, E3 +442653.903}
SPL {X  -161.904, Y  +363.251, Z    +0.000, E1   +14.606, E3 +442683.698}
SPL {X  -162.745, Y  +375.561, Z    +0.000, E1    +7.538, E3 +442683.895}
SPL {X  -162.820, Y  +385.424, Z    +0.000, E1    +1.080, E3 +442684.789}
SPL {X  -162.820, Y  +389.940, Z    +0.000, E1    -2.281, E3 +442687.666}
SPL {X  -162.820, Y  +396.652, Z    +0.000, E1    -7.520, E3 +442687.244}
SPL {X  -162.820, Y  +406.605, Z    +0.000, E1   -16.760, E3 +442679.721}
SPL {X  -162.820, Y  +418.675, Z    +0.000, E1   -22.201, E3 +442705.970}
SPL {X  -162.820, Y  +425.113, Z    +0.000, E1   -25.243, E3 +442714.906}
SPL {X  -162.820, Y  +441.937, Z    +0.000, E1   -31.578, E3 +442736.984}
ENDSPLINE

SPLINE
SPL {X  -162.820, Y  +437.771, Z    +0.000, E1   -26.555, E3 +442756.084}
ENDSPLINE

SPLINE
SPL {X  -162.820, Y  +439.120, Z    +0.000, E1   -25.352, E3 +442770.628}
SPL {X  -162.820, Y  +441.593, Z    +0.000, E1   -25.391, E3 +442781.179}
SPL {X  -162.820, Y  +444.317, Z    +0.000, E1   -25.492, E3 +442792.361}
SPL {X  -162.820, Y  +446.544, Z    +0.000, E1   -25.427, E3 +442802.530}
SPL {X  -162.820, Y  +448.500, Z    +0.000, E1   -25.425, E3 +442811.132}
SPL {X  -162.820, Y  +451.056, Z    +0.000, E1   -25.443, E3 +442822.239}
SPL {X  -162.820, Y  +454.662, Z    +0.000, E1   -25.474, E3 +442837.984}
SPL {X  -162.820, Y  +458.079, Z    +0.000, E1   -25.369, E3 +442853.563}
SPL {X  -162.820, Y  +460.719, Z    +0.000, E1   -25.411, E3 +442864.821}
SPL {X  -162.820, Y  +463.419, Z    +0.000, E1   -25.510, E3 +442875.859}
SPL {X  -162.820, Y  +466.458, Z    +0.000, E1   -25.433, E3 +442889.914}
SPL {X  -162.820, Y  +470.010, Z    +0.000, E1   -25.445, E3 +442905.283}
SPL {X  -162.820, Y  +472.345, Z    +0.000, E1   -25.448, E3 +442915.369}
SPL {X  -162.820, Y  +475.191, Z    +0.000, E1   -25.489, E3 +442927.731}
SPL {X  -162.820, Y  +478.461, Z    +0.000, E1   -25.410, E3 +442942.501}
SPL {X  -162.820, Y  +480.780, Z    +0.000, E1   -25.447, E3 +442952.363}
SPL {X  -162.820, Y  +483.622, Z    +0.000, E1   -25.381, E3 +442965.404}
SPL {X  -162.820, Y  +486.874, Z    +0.000, E1   -25.478, E3 +442978.866}
SPL {X  -162.820, Y  +490.287, Z    +0.000, E1   -25.463, E3 +442994.085}
SPL {X  -162.820, Y  +494.454, Z    +0.000, E1   -25.465, E3 +443012.316}
SPL {X  -162.820, Y  +498.644, Z    +0.000, E1   -25.463, E3 +443030.693}
SPL {X  -162.820, Y  +502.845, Z    +0.000, E1   -25.458, E3 +443049.126}
SPL {X  -162.820, Y  +506.050, Z    +0.000, E1   -25.420, E3 +443063.266}
SPL {X  -162.820, Y  +508.346, Z    +0.000, E1   -25.444, E3 +443073.114}
SPL {X  -162.820, Y  +511.422, Z    +0.000, E1   -25.445, E3 +443086.775}
SPL {X  -162.820, Y  +515.039, Z    +0.000, E1   -25.452, E3 +443102.456}
SPL {X  -162.820, Y  +517.481, Z    +0.000, E1   -25.432, E3 +443113.190}
SPL {X  -162.820, Y  +519.134, Z    +0.000, E1   -25.366, E3 +443120.937}
SPL {X  -162.820, Y  +521.486, Z    +0.000, E1   -25.382, E3 +443131.233}
SPL {X  -162.820, Y  +525.073, Z    +0.000, E1   -25.512, E3 +443146.039}
SPL {X  -162.820, Y  +527.738, Z    +0.000, E1   -25.438, E3 +443158.087}
SPL {X  -162.820, Y  +530.432, Z    +0.000, E1   -25.477, E3 +443169.664}
SPL {X  -162.820, Y  +534.051, Z    +0.000, E1   -25.484, E3 +443185.541}
SPL {X  -162.820, Y  +537.226, Z    +0.000, E1   -25.378, E3 +443200.111}
SPL {X  -162.820, Y  +539.521, Z    +0.000, E1   -25.386, E3 +443210.069}
SPL {X  -162.820, Y  +542.667, Z    +0.000, E1   -25.474, E3 +443223.394}
SPL {X  -162.820, Y  +546.125, Z    +0.000, E1   -25.505, E3 +443238.119}
SPL {X  -162.820, Y  +548.232, Z    +0.000, E1   -25.424, E3 +443247.881}
SPL {X  -162.820, Y  +550.399, Z    +0.000, E1   -25.424, E3 +443257.432}
SPL {X  -162.820, Y  +553.157, Z    +0.000, E1   -25.443, E3 +443269.407}
SPL {X  -162.820, Y  +556.150, Z    +0.000, E1   -25.445, E3 +443282.496}
SPL {X  -162.820, Y  +559.215, Z    +0.000, E1   -25.460, E3 +443295.798}
SPL {X  -162.820, Y  +562.125, Z    +0.000, E1   -25.434, E3 +443308.718}
SPL {X  -162.820, Y  +564.880, Z    +0.000, E1   -25.448, E3 +443320.672}
SPL {X  -162.820, Y  +568.326, Z    +0.000, E1   -25.470, E3 +443335.732}
SPL {X  -162.820, Y  +571.303, Z    +0.000, E1   -25.427, E3 +443348.905}
SPL {X  -162.820, Y  +574.067, Z    +0.000, E1   -25.459, E3 +443360.844}
SPL {X  -162.820, Y  +576.597, Z    +0.000, E1   -25.400, E3 +443372.315}
SPL {X  -162.820, Y  +580.038, Z    +0.000, E1   -25.473, E3 +443387.010}
SPL {X  -162.820, Y  +583.044, Z    +0.000, E1   -25.450, E3 +443400.134}
SPL {X  -162.820, Y  +585.512, Z    +0.000, E1   -25.448, E3 +443411.029}
SPL {X  -162.820, Y  +588.371, Z    +0.000, E1   -25.460, E3 +443423.415}
SPL {X  -162.820, Y  +590.476, Z    +0.000, E1   -25.398, E3 +443433.056}
SPL {X  -162.820, Y  +593.604, Z    +0.000, E1   -25.477, E3 +443446.335}
SPL {X  -162.820, Y  +596.868, Z    +0.000, E1   -25.461, E3 +443460.600}
SPL {X  -162.820, Y  +599.135, Z    +0.000, E1   -25.398, E3 +443470.969}
SPL {X  -162.820, Y  +601.296, Z    +0.000, E1   -25.399, E3 +443480.451}
SPL {X  -162.820, Y  +604.526, Z    +0.000, E1   -25.502, E3 +443493.944}
SPL {X  -162.820, Y  +607.811, Z    +0.000, E1   -25.507, E3 +443508.159}
SPL {X  -162.820, Y  +610.517, Z    +0.000, E1   -25.412, E3 +443520.721}
SPL {X  -162.820, Y  +613.762, Z    +0.000, E1   -25.472, E3 +443534.528}
SPL {X  -162.820, Y  +616.216, Z    +0.000, E1   -25.419, E3 +443545.524}
SPL {X  -162.820, Y  +618.995, Z    +0.000, E1   -25.483, E3 +443557.373}
SPL {X  -162.820, Y  +622.118, Z    +0.000, E1   -25.492, E3 +443570.838}
SPL {X  -162.820, Y  +624.430, Z    +0.000, E1   -25.475, E3 +443581.059}
SPL {X  -162.820, Y  +626.570, Z    +0.000, E1   -25.441, E3 +443590.660}
SPL {X  -162.820, Y  +628.902, Z    +0.000, E1   -25.449, E3 +443600.840}
SPL {X  -162.820, Y  +631.177, Z    +0.000, E1   -25.467, E3 +443610.671}
SPL {X  -162.820, Y  +633.994, Z    +0.000, E1   -25.503, E3 +443622.718}
SPL {X  -162.820, Y  +636.469, Z    +0.000, E1   -25.465, E3 +443633.761}
SPL {X  -162.820, Y  +638.486, Z    +0.000, E1   -25.456, E3 +443642.679}
SPL {X  -162.820, Y  +640.803, Z    +0.000, E1   -25.462, E3 +443652.740}
SPL {X  -162.820, Y  +643.028, Z    +0.000, E1   -25.494, E3 +443662.250}
SPL {X  -162.820, Y  +646.519, Z    +0.000, E1   -25.551, E3 +443677.232}
SPL {X  -162.820, Y  +649.837, Z    +0.000, E1   -25.446, E3 +443692.356}
SPL {X  -162.820, Y  +652.810, Z    +0.000, E1   -25.497, E3 +443704.999}
SPL {X  -162.820, Y  +655.214, Z    +0.000, E1   -25.485, E3 +443715.502}
SPL {X  -162.820, Y  +657.616, Z    +0.000, E1   -25.511, E3 +443725.856}
SPL {X  -162.820, Y  +660.851, Z    +0.000, E1   -25.520, E3 +443739.999}
SPL {X  -162.820, Y  +663.853, Z    +0.000, E1   -25.496, E3 +443753.180}
SPL {X  -162.820, Y  +667.253, Z    +0.000, E1   -25.483, E3 +443768.353}
SPL {X  -162.820, Y  +671.102, Z    +0.000, E1   -25.514, E3 +443784.803}
SPL {X  -162.820, Y  +673.648, Z    +0.000, E1   -25.431, E3 +443796.470}
SPL {X  -162.796, Y  +676.319, Z    +0.000, E1   -25.526, E3 +443807.479}
SPL {X  -162.739, Y  +678.625, Z    +0.000, E1   -25.423, E3 +443818.271}
SPL {X  -162.669, Y  +680.515, Z    +0.000, E1   -25.398, E3 +443826.725}
SPL {X  -162.545, Y  +682.952, Z    +0.000, E1   -25.510, E3 +443836.587}
SPL {X  -162.381, Y  +685.455, Z    +0.000, E1   -25.410, E3 +443848.273}
SPL {X  -162.194, Y  +687.760, Z    +0.000, E1   -25.360, E3 +443858.709}
SPL {X  -161.987, Y  +689.945, Z    +0.000, E1   -25.406, E3 +443867.862}
SPL {X  -161.711, Y  +692.468, Z    +0.000, E1   -25.300, E3 +443879.860}
SPL {X  -160.732, Y  +699.494, Z    +0.000, E1   -27.462, E3 +443893.333}
SPL {X  -157.189, Y  +715.948, Z    +0.000, E1   -34.218, E3 +443905.491}
ENDSPLINE

SPLINE
SPL {X  -157.848, Y  +713.428, Z    +0.000, E1   -28.857, E3 +443939.630}
SPL {X  -161.035, Y  +697.541, Z    +0.000, E1   -20.899, E3 +443940.149}
SPL {X  -161.689, Y  +692.657, Z    +0.000, E1   -15.656, E3 +443980.232}
SPL {X  -162.807, Y  +675.545, Z    +0.000, E1    -5.787, E3 +443975.732}
ENDSPLINE

SPLINE
SPL {X  -162.791, Y  +676.574, Z    +0.000, E1    -6.127, E3 +443988.834}
ENDSPLINE

SPLINE
SPL {X  -162.820, Y  +664.716, Z    +0.000, E1    +1.705, E3 +443977.708}
SPL {X  -162.820, Y  +658.484, Z    +0.000, E1    +6.336, E3 +443984.185}
SPL {X  -162.820, Y  +640.102, Z    +0.000, E1   +22.409, E3 +443978.923}
SPL {X  -162.820, Y  +633.503, Z    +0.000, E1   +21.975, E3 +444011.160}
SPL {X  -162.820, Y  +611.299, Z    +0.000, E1   +31.088, E3 +444039.273}
ENDSPLINE

SPLINE
SPL {X  -162.820, Y  +618.877, Z    +0.000, E1   +25.259, E3 +444050.767}
ENDSPLINE

SPLINE
SPL {X  -162.820, Y  +617.582, Z    +0.000, E1   +24.552, E3 +444062.144}
SPL {X  -162.820, Y  +614.716, Z    +0.000, E1   +24.535, E3 +444075.355}
SPL {X  -162.820, Y  +611.754, Z    +0.000, E1   +24.563, E3 +444088.643}
SPL {X  -162.820, Y  +608.970, Z    +0.000, E1   +24.542, E3 +444101.483}
SPL {X  -162.820, Y  +606.285, Z    +0.000, E1   +24.533, E3 +444113.819}
SPL {X  -162.820, Y  +603.509, Z    +0.000, E1   +24.546, E3 +444126.356}
SPL {X  -162.820, Y  +600.818, Z    +0.000, E1   +24.590, E3 +444138.279}
SPL {X  -162.820, Y  +598.053, Z    +0.000, E1   +24.547, E3 +444151.262}
SPL {X  -162.820, Y  +595.188, Z    +0.000, E1   +24.538, E3 +444164.351}
SPL {X  -162.820, Y  +592.738, Z    +0.000, E1   +24.551, E3 +444175.399}
SPL {X  -162.820, Y  +590.118, Z    +0.000, E1   +24.544, E3 +444187.458}
SPL {X  -162.820, Y  +587.204, Z    +0.000, E1   +24.592, E3 +444200.335}
SPL {X  -162.820, Y  +584.766, Z    +0.000, E1   +24.499, E3 +444212.168}
SPL {X  -162.820, Y  +581.896, Z    +0.000, E1   +24.528, E3 +444225.110}
SPL {X  -162.820, Y  +578.588, Z    +0.000, E1   +24.598, E3 +444239.661}
SPL {X  -162.820, Y  +575.299, Z    +0.000, E1   +24.560, E3 +444254.958}
SPL {X  -162.820, Y  +572.074, Z    +0.000, E1   +24.505, E3 +444270.097}
SPL {X  -162.820, Y  +568.309, Z    +0.000, E1   +24.589, E3 +444286.724}
SPL {X  -162.820, Y  +564.977, Z    +0.000, E1   +24.571, E3 +444301.896}
SPL {X  -162.820, Y  +562.356, Z    +0.000, E1   +24.575, E3 +444313.795}
SPL {X  -162.820, Y  +560.119, Z    +0.000, E1   +24.506, E3 +444324.484}
SPL {X  -162.820, Y  +558.093, Z    +0.000, E1   +24.537, E3 +444333.502}
SPL {X  -162.820, Y  +555.584, Z    +0.000, E1   +24.559, E3 +444344.814}
SPL {X  -162.820, Y  +552.867, Z    +0.000, E1   +24.583, E3 +444357.009}
SPL {X  -162.820, Y  +549.589, Z    +0.000, E1   +24.547, E3 +444372.376}
SPL {X  -162.820, Y  +545.742, Z    +0.000, E1   +24.577, E3 +444389.662}
SPL {X  -162.820, Y  +542.142, Z    +0.000, E1   +24.582, E3 +444406.016}
SPL {X  -162.820, Y  +538.903, Z    +0.000, E1   +24.519, E3 +444421.231}
SPL {X  -162.820, Y  +536.451, Z    +0.000, E1   +24.519, E3 +444432.311}
SPL {X  -162.820, Y  +534.025, Z    +0.000, E1   +24.589, E3 +444442.912}
SPL {X  -162.820, Y  +531.527, Z    +0.000, E1   +24.582, E3 +444454.297}
SPL {X  -162.820, Y  +529.165, Z    +0.000, E1   +24.521, E3 +444465.546}
SPL {X  -162.820, Y  +525.802, Z    +0.000, E1   +24.585, E3 +444480.566}
SPL {X  -162.820, Y  +521.731, Z    +0.000, E1   +24.542, E3 +444499.502}
SPL {X  -162.820, Y  +518.185, Z    +0.000, E1   +24.561, E3 +444515.374}
SPL {X  -162.820, Y  +508.728, Z    +0.000, E1   +28.484, E3 +444525.914}
SPL {X  -162.820, Y  +500.664, Z    +0.000, E1   +31.476, E3 +444534.578}
SPL {X  -162.820, Y  +499.290, Z    +0.000, E1   +30.657, E3 +444544.860}
SPL {X  -162.820, Y  +497.251, Z    +0.000, E1   +29.634, E3 +444559.336}
SPL {X  -162.820, Y  +495.647, Z    +0.000, E1   +28.606, E3 +444572.212}
SPL {X  -162.820, Y  +494.678, Z    +0.000, E1   +27.647, E3 +444582.913}
SPL {X  -162.820, Y  +493.757, Z    +0.000, E1   +26.462, E3 +444595.273}
SPL {X  -162.820, Y  +491.420, Z    +0.000, E1   +25.780, E3 +444610.534}
SPL {X  -162.820, Y  +487.351, Z    +0.000, E1   +25.663, E3 +444629.051}
SPL {X  -162.820, Y  +484.247, Z    +0.000, E1   +25.651, E3 +444642.377}
SPL {X  -162.820, Y  +482.092, Z    +0.000, E1   +25.593, E3 +444652.204}
SPL {X  -162.820, Y  +479.578, Z    +0.000, E1   +25.634, E3 +444662.847}
SPL {X  -162.820, Y  +477.137, Z    +0.000, E1   +25.632, E3 +444673.426}
SPL {X  -162.820, Y  +473.770, Z    +0.000, E1   +25.664, E3 +444687.972}
SPL {X  -162.820, Y  +469.694, Z    +0.000, E1   +25.657, E3 +444705.703}
SPL {X  -162.820, Y  +465.727, Z    +0.000, E1   +25.676, E3 +444722.746}
SPL {X  -162.820, Y  +461.675, Z    +0.000, E1   +25.655, E3 +444740.552}
SPL {X  -162.820, Y  +457.479, Z    +0.000, E1   +25.656, E3 +444758.732}
SPL {X  -162.820, Y  +453.678, Z    +0.000, E1   +25.652, E3 +444775.184}
SPL {X  -162.820, Y  +450.466, Z    +0.000, E1   +25.644, E3 +444789.129}
SPL {X  -162.820, Y  +447.822, Z    +0.000, E1   +25.664, E3 +444800.387}
SPL {X  -162.820, Y  +444.499, Z    +0.000, E1   +25.673, E3 +444814.958}
SPL {X  -162.820, Y  +440.857, Z    +0.000, E1   +25.614, E3 +444831.066}
SPL {X  -162.820, Y  +437.636, Z    +0.000, E1   +25.597, E3 +444845.230}
SPL {X  -162.820, Y  +434.768, Z    +0.000, E1   +25.655, E3 +444857.131}
SPL {X  -162.820, Y  +431.823, Z    +0.000, E1   +25.651, E3 +444870.130}
SPL {X  -162.820, Y  +427.740, Z    +0.000, E1   +25.667, E3 +444887.759}
SPL {X  -162.820, Y  +423.655, Z    +0.000, E1   +25.628, E3 +444905.783}
SPL {X  -162.820, Y  +419.407, Z    +0.000, E1   +25.665, E3 +444923.975}
SPL {X  -162.820, Y  +415.900, Z    +0.000, E1   +25.638, E3 +444939.245}
SPL {X  -162.820, Y  +413.088, Z    +0.000, E1   +25.644, E3 +444951.401}
SPL {X  -162.820, Y  +410.320, Z    +0.000, E1   +25.604, E3 +444963.720}
SPL {X  -162.820, Y  +407.487, Z    +0.000, E1   +25.617, E3 +444975.927}
SPL {X  -162.820, Y  +405.108, Z    +0.000, E1   +25.535, E3 +444986.895}
SPL {X  -162.820, Y  +401.373, Z    +0.000, E1   +25.736, E3 +445001.732}
SPL {X  -162.820, Y  +397.357, Z    +0.000, E1   +25.652, E3 +445019.802}
SPL {X  -162.820, Y  +393.659, Z    +0.000, E1   +25.666, E3 +445035.602}
SPL {X  -162.820, Y  +390.679, Z    +0.000, E1   +25.624, E3 +445048.845}
SPL {X  -162.820, Y  +387.939, Z    +0.000, E1   +25.627, E3 +445060.705}
SPL {X  -162.820, Y  +384.398, Z    +0.000, E1   +25.707, E3 +445075.603}
SPL {X  -162.820, Y  +380.448, Z    +0.000, E1   +25.674, E3 +445092.966}
SPL {X  -162.785, Y  +377.106, Z    +0.000, E1   +25.598, E3 +445107.911}
SPL {X  -162.709, Y  +374.484, Z    +0.000, E1   +25.711, E3 +445118.362}
SPL {X  -162.623, Y  +372.485, Z    +0.000, E1   +25.631, E3 +445127.642}
SPL {X  -162.487, Y  +370.088, Z    +0.000, E1   +25.525, E3 +445138.896}
SPL {X  -162.243, Y  +366.801, Z    +0.000, E1   +25.618, E3 +445152.536}
SPL {X  -161.977, Y  +363.953, Z    +0.000, E1   +25.528, E3 +445165.463}
SPL {X  -161.695, Y  +361.389, Z    +0.000, E1   +25.445, E3 +445177.278}
SPL {X  -161.364, Y  +358.774, Z    +0.000, E1   +25.454, E3 +445188.479}
SPL {X  -160.939, Y  +355.820, Z    +0.000, E1   +26.179, E3 +445195.697}
SPL {X  -155.035, Y  +330.756, Z    +0.000, E1   +37.918, E3 +445202.031}
SPL {X  -153.918, Y  +327.401, Z    +0.000, E1   +34.677, E3 +445237.331}
ENDSPLINE

SPLINE
SPL {X  -159.701, Y  +348.785, Z    +0.000, E1   +24.361, E3 +445244.812}
SPL {X  -161.904, Y  +363.251, Z    +0.000, E1   +14.606, E3 +445274.607}
SPL {X  -162.745, Y  +375.561, Z    +0.000, E1    +7.538, E3 +445274.804}
SPL {X  -162.820, Y  +385.424, Z    +0.000, E1    +1.080, E3 +445275.698}
SPL {X  -162.820, Y  +389.940, Z    +0.000, E1    -2.281, E3 +445278.575}
SPL {X  -162.820, Y  +396.652, Z    +0.000, E1    -7.520, E3 +445278.153}
SPL {X  -162.820, Y  +406.605, Z    +0.000, E1   -16.760, E3 +445270.630}
SPL {X  -162.820, Y  +420.013, Z    +0.000, E1   -22.833, E3 +445298.751}
SPL {X  -162.820, Y  +442.075, Z    +0.000, E1   -31.090, E3 +445331.537}
ENDSPLINE

SPLINE
SPL {X  -162.820, Y  +436.680, Z    +0.000, E1   -26.151, E3 +445344.841}
ENDSPLINE

SPLINE
SPL {X  -162.820, Y  +438.487, Z    +0.000, E1   -25.409, E3 +445358.480}
SPL {X  -162.820, Y  +441.593, Z    +0.000, E1   -25.391, E3 +445372.088}
SPL {X  -162.820, Y  +444.317, Z    +0.000, E1   -25.492, E3 +445383.270}
SPL {X  -162.820, Y  +446.544, Z    +0.000, E1   -25.427, E3 +445393.439}
SPL {X  -162.820, Y  +448.500, Z    +0.000, E1   -25.425, E3 +445402.041}
SPL {X  -162.820, Y  +451.056, Z    +0.000, E1   -25.443, E3 +445413.148}
SPL {X  -162.820, Y  +454.662, Z    +0.000, E1   -25.474, E3 +445428.893}
SPL {X  -162.820, Y  +458.079, Z    +0.000, E1   -25.369, E3 +445444.472}
SPL {X  -162.820, Y  +460.719, Z    +0.000, E1   -25.411, E3 +445455.730}
SPL {X  -162.820, Y  +463.419, Z    +0.000, E1   -25.510, E3 +445466.768}
SPL {X  -162.820, Y  +466.458, Z    +0.000, E1   -25.433, E3 +445480.823}
SPL {X  -162.820, Y  +470.010, Z    +0.000, E1   -25.445, E3 +445496.192}
SPL {X  -162.820, Y  +472.345, Z    +0.000, E1   -25.448, E3 +445506.278}
SPL {X  -162.820, Y  +475.191, Z    +0.000, E1   -25.489, E3 +445518.641}
SPL {X  -162.820, Y  +478.461, Z    +0.000, E1   -25.410, E3 +445533.410}
SPL {X  -162.820, Y  +480.780, Z    +0.000, E1   -25.447, E3 +445543.272}
SPL {X  -162.820, Y  +483.622, Z    +0.000, E1   -25.381, E3 +445556.314}
SPL {X  -162.820, Y  +487.570, Z    +0.000, E1   -25.482, E3 +445572.952}
SPL {X  -162.820, Y  +491.017, Z    +0.000, E1   -25.445, E3 +445588.166}
SPL {X  -162.820, Y  +493.705, Z    +0.000, E1   -25.443, E3 +445599.951}
SPL {X  -162.820, Y  +497.247, Z    +0.000, E1   -25.470, E3 +445615.413}
SPL {X  -162.820, Y  +501.343, Z    +0.000, E1   -25.435, E3 +445633.612}
SPL {X  -162.820, Y  +505.370, Z    +0.000, E1   -25.456, E3 +445651.075}
SPL {X  -162.820, Y  +509.412, Z    +0.000, E1   -25.458, E3 +445668.798}
SPL {X  -162.820, Y  +512.406, Z    +0.000, E1   -25.425, E3 +445681.954}
SPL {X  -162.820, Y  +515.039, Z    +0.000, E1   -25.452, E3 +445693.365}
SPL {X  -162.820, Y  +518.350, Z    +0.000, E1   -25.425, E3 +445708.114}
SPL {X  -162.820, Y  +521.486, Z    +0.000, E1   -25.382, E3 +445722.142}
SPL {X  -162.820, Y  +524.180, Z    +0.000, E1   -25.495, E3 +445733.014}
SPL {X  -162.820, Y  +527.020, Z    +0.000, E1   -25.477, E3 +445745.707}
SPL {X  -162.820, Y  +529.670, Z    +0.000, E1   -25.472, E3 +445757.165}
SPL {X  -162.820, Y  +532.006, Z    +0.000, E1   -25.455, E3 +445767.622}
SPL {X  -162.820, Y  +534.806, Z    +0.000, E1   -25.465, E3 +445779.738}
SPL {X  -162.820, Y  +537.226, Z    +0.000, E1   -25.378, E3 +445791.020}
SPL {X  -162.820, Y  +540.345, Z    +0.000, E1   -25.451, E3 +445804.201}
SPL {X  -162.820, Y  +543.279, Z    +0.000, E1   -25.419, E3 +445817.234}
SPL {X  -162.820, Y  +546.125, Z    +0.000, E1   -25.505, E3 +445829.028}
SPL {X  -162.820, Y  +549.578, Z    +0.000, E1   -25.462, E3 +445844.652}
SPL {X  -162.820, Y  +553.157, Z    +0.000, E1   -25.443, E3 +445860.316}
SPL {X  -162.820, Y  +556.965, Z    +0.000, E1   -25.478, E3 +445876.908}
SPL {X  -162.820, Y  +561.429, Z    +0.000, E1   -25.478, E3 +445896.427}
SPL {X  -162.820, Y  +565.606, Z    +0.000, E1   -25.468, E3 +445914.757}
SPL {X  -162.820, Y  +568.974, Z    +0.000, E1   -25.453, E3 +445929.467}
SPL {X  -162.820, Y  +571.303, Z    +0.000, E1   -25.427, E3 +445939.814}
SPL {X  -162.820, Y  +574.067, Z    +0.000, E1   -25.459, E3 +445951.753}
SPL {X  -162.820, Y  +576.597, Z    +0.000, E1   -25.400, E3 +445963.224}
SPL {X  -162.820, Y  +580.038, Z    +0.000, E1   -25.473, E3 +445977.919}
SPL {X  -162.820, Y  +583.044, Z    +0.000, E1   -25.450, E3 +445991.043}
SPL {X  -162.820, Y  +585.512, Z    +0.000, E1   -25.448, E3 +446001.938}
SPL {X  -162.820, Y  +588.371, Z    +0.000, E1   -25.460, E3 +446014.324}
SPL {X  -162.820, Y  +591.246, Z    +0.000, E1   -25.415, E3 +446027.343}
SPL {X  -162.820, Y  +594.339, Z    +0.000, E1   -25.487, E3 +446040.246}
SPL {X  -162.820, Y  +596.868, Z    +0.000, E1   -25.461, E3 +446051.509}
SPL {X  -162.820, Y  +600.326, Z    +0.000, E1   -25.438, E3 +446067.030}
SPL {X  -162.820, Y  +604.526, Z    +0.000, E1   -25.502, E3 +446084.853}
SPL {X  -162.820, Y  +607.811, Z    +0.000, E1   -25.507, E3 +446099.068}
SPL {X  -162.820, Y  +610.517, Z    +0.000, E1   -25.412, E3 +446111.630}
SPL {X  -162.820, Y  +613.762, Z    +0.000, E1   -25.472, E3 +446125.437}
SPL {X  -162.820, Y  +617.275, Z    +0.000, E1   -25.466, E3 +446140.876}
SPL {X  -162.820, Y  +621.264, Z    +0.000, E1   -25.514, E3 +446158.037}
SPL {X  -162.820, Y  +624.430, Z    +0.000, E1   -25.475, E3 +446171.968}
SPL {X  -162.820, Y  +626.570, Z    +0.000, E1   -25.441, E3 +446181.569}
SPL {X  -162.820, Y  +628.902, Z    +0.000, E1   -25.449, E3 +446191.749}
SPL {X  -162.820, Y  +631.177, Z    +0.000, E1   -25.467, E3 +446201.580}
SPL {X  -162.820, Y  +633.994, Z    +0.000, E1   -25.503, E3 +446213.627}
SPL {X  -162.820, Y  +637.619, Z    +0.000, E1   -25.497, E3 +446229.687}
SPL {X  -162.820, Y  +640.803, Z    +0.000, E1   -25.462, E3 +446243.649}
SPL {X  -162.820, Y  +643.028, Z    +0.000, E1   -25.494, E3 +446253.159}
SPL {X  -162.820, Y  +646.519, Z    +0.000, E1   -25.551, E3 +446268.141}
SPL {X  -162.820, Y  +649.837, Z    +0.000, E1   -25.446, E3 +446283.265}
SPL {X  -162.820, Y  +652.810, Z    +0.000, E1   -25.497, E3 +446295.908}
SPL {X  -162.820, Y  +655.214, Z    +0.000, E1   -25.485, E3 +446306.411}
SPL {X  -162.820, Y  +657.616, Z    +0.000, E1   -25.511, E3 +446316.765}
SPL {X  -162.820, Y  +660.007, Z    +0.000, E1   -25.550, E3 +446326.826}
SPL {X  -162.820, Y  +662.980, Z    +0.000, E1   -25.505, E3 +446340.385}
SPL {X  -162.820, Y  +667.253, Z    +0.000, E1   -25.483, E3 +446359.262}
SPL {X  -162.820, Y  +671.102, Z    +0.000, E1   -25.514, E3 +446375.712}
SPL {X  -162.820, Y  +673.648, Z    +0.000, E1   -25.431, E3 +446387.379}
SPL {X  -162.796, Y  +676.319, Z    +0.000, E1   -25.526, E3 +446398.388}
SPL {X  -162.707, Y  +679.552, Z    +0.000, E1   -25.443, E3 +446413.263}
SPL {X  -162.545, Y  +682.952, Z    +0.000, E1   -25.510, E3 +446427.496}
SPL {X  -162.381, Y  +685.455, Z    +0.000, E1   -25.410, E3 +446439.182}
SPL {X  -162.102, Y  +688.774, Z    +0.000, E1   -25.417, E3 +446453.797}
SPL {X  -161.711, Y  +692.468, Z    +0.000, E1   -25.300, E3 +446470.769}
SPL {X  -161.141, Y  +696.825, Z    +0.000, E1   -26.170, E3 +446482.904}
SPL {X  -157.976, Y  +712.921, Z    +0.000, E1   -33.197, E3 +446493.444}
ENDSPLINE

SPLINE
SPL {X  -160.738, Y  +699.453, Z    +0.000, E1   -21.994, E3 +446531.071}
SPL {X  -161.689, Y  +692.657, Z    +0.000, E1   -15.656, E3 +446571.141}
SPL {X  -162.807, Y  +675.545, Z    +0.000, E1    -5.787, E3 +446566.641}
ENDSPLINE

SPLINE
SPL {X  -162.791, Y  +676.574, Z    +0.000, E1    -6.127, E3 +446579.743}
ENDSPLINE

SPLINE
SPL {X  -162.820, Y  +664.716, Z    +0.000, E1    +1.705, E3 +446568.617}
SPL {X  -162.820, Y  +658.484, Z    +0.000, E1    +6.336, E3 +446575.094}
SPL {X  -162.820, Y  +640.102, Z    +0.000, E1   +22.409, E3 +446569.832}
SPL {X  -162.820, Y  +633.503, Z    +0.000, E1   +21.975, E3 +446602.069}
SPL {X  -162.820, Y  +611.299, Z    +0.000, E1   +31.088, E3 +446630.182}
ENDSPLINE

SPLINE
SPL {X  -162.820, Y  +618.877, Z    +0.000, E1   +25.259, E3 +446641.676}
ENDSPLINE

SPLINE
SPL {X  -162.820, Y  +617.582, Z    +0.000, E1   +24.552, E3 +446653.053}
SPL {X  -162.820, Y  +614.716, Z    +0.000, E1   +24.535, E3 +446666.264}
SPL {X  -162.820, Y  +611.754, Z    +0.000, E1   +24.563, E3 +446679.552}
SPL {X  -162.820, Y  +608.970, Z    +0.000, E1   +24.542, E3 +446692.393}
SPL {X  -162.820, Y  +606.285, Z    +0.000, E1   +24.533, E3 +446704.728}
SPL {X  -162.820, Y  +603.509, Z    +0.000, E1   +24.546, E3 +446717.265}
SPL {X  -162.820, Y  +600.818, Z    +0.000, E1   +24.590, E3 +446729.188}
SPL {X  -162.820, Y  +598.053, Z    +0.000, E1   +24.547, E3 +446742.171}
SPL {X  -162.820, Y  +595.188, Z    +0.000, E1   +24.538, E3 +446755.260}
SPL {X  -162.820, Y  +592.738, Z    +0.000, E1   +24.551, E3 +446766.308}
SPL {X  -162.820, Y  +590.118, Z    +0.000, E1   +24.544, E3 +446778.367}
SPL {X  -162.820, Y  +587.204, Z    +0.000, E1   +24.592, E3 +446791.244}
SPL {X  -162.820, Y  +584.193, Z    +0.000, E1   +24.484, E3 +446805.954}
SPL {X  -162.820, Y  +580.163, Z    +0.000, E1   +24.634, E3 +446823.189}
SPL {X  -162.820, Y  +576.848, Z    +0.000, E1   +24.543, E3 +446838.904}
SPL {X  -162.820, Y  +574.433, Z    +0.000, E1   +24.551, E3 +446849.735}
SPL {X  -162.820, Y  +572.074, Z    +0.000, E1   +24.505, E3 +446861.006}
SPL {X  -162.820, Y  +569.438, Z    +0.000, E1   +24.562, E3 +446872.465}
SPL {X  -162.820, Y  +567.494, Z    +0.000, E1   +24.547, E3 +446881.475}
SPL {X  -162.820, Y  +564.977, Z    +0.000, E1   +24.571, E3 +446892.806}
SPL {X  -162.820, Y  +562.356, Z    +0.000, E1   +24.575, E3 +446904.704}
SPL {X  -162.820, Y  +560.119, Z    +0.000, E1   +24.506, E3 +446915.393}
SPL {X  -162.820, Y  +558.093, Z    +0.000, E1   +24.537, E3 +446924.411}
SPL {X  -162.820, Y  +555.584, Z    +0.000, E1   +24.559, E3 +446935.723}
SPL {X  -162.820, Y  +552.169, Z    +0.000, E1   +24.581, E3 +446951.292}
SPL {X  -162.820, Y  +548.932, Z    +0.000, E1   +24.540, E3 +446966.193}
SPL {X  -162.820, Y  +545.742, Z    +0.000, E1   +24.577, E3 +446980.571}
SPL {X  -162.820, Y  +542.142, Z    +0.000, E1   +24.582, E3 +446996.925}
SPL {X  -162.820, Y  +538.903, Z    +0.000, E1   +24.519, E3 +447012.140}
SPL {X  -162.820, Y  +536.451, Z    +0.000, E1   +24.519, E3 +447023.220}
SPL {X  -162.820, Y  +534.025, Z    +0.000, E1   +24.589, E3 +447033.821}
SPL {X  -162.820, Y  +531.527, Z    +0.000, E1   +24.582, E3 +447045.206}
SPL {X  -162.820, Y  +529.165, Z    +0.000, E1   +24.521, E3 +447056.455}
SPL {X  -162.820, Y  +526.822, Z    +0.000, E1   +24.559, E3 +447066.818}
SPL {X  -162.820, Y  +524.112, Z    +0.000, E1   +24.542, E3 +447079.436}
SPL {X  -162.820, Y  +521.048, Z    +0.000, E1   +24.515, E3 +447093.572}
SPL {X  -162.820, Y  +518.185, Z    +0.000, E1   +24.561, E3 +447106.283}
SPL {X  -162.820, Y  +508.728, Z    +0.000, E1   +28.484, E3 +447116.823}
SPL {X  -162.820, Y  +500.664, Z    +0.000, E1   +31.476, E3 +447125.487}
SPL {X  -162.820, Y  +499.290, Z    +0.000, E1   +30.657, E3 +447135.769}
SPL {X  -162.820, Y  +497.251, Z    +0.000, E1   +29.634, E3 +447150.245}
SPL {X  -162.820, Y  +495.647, Z    +0.000, E1   +28.606, E3 +447163.121}
SPL {X  -162.820, Y  +494.678, Z    +0.000, E1   +27.647, E3 +447173.822}
SPL {X  -162.820, Y  +493.757, Z    +0.000, E1   +26.462, E3 +447186.182}
SPL {X  -162.820, Y  +492.330, Z    +0.000, E1   +25.953, E3 +447195.936}
SPL {X  -162.820, Y  +489.800, Z    +0.000, E1   +25.653, E3 +447209.398}
SPL {X  -162.820, Y  +485.392, Z    +0.000, E1   +25.667, E3 +447228.425}
SPL {X  -162.820, Y  +482.092, Z    +0.000, E1   +25.593, E3 +447243.113}
SPL {X  -162.820, Y  +479.578, Z    +0.000, E1   +25.634, E3 +447253.756}
SPL {X  -162.820, Y  +477.137, Z    +0.000, E1   +25.632, E3 +447264.335}
SPL {X  -162.820, Y  +473.770, Z    +0.000, E1   +25.664, E3 +447278.881}
SPL {X  -162.820, Y  +469.694, Z    +0.000, E1   +25.657, E3 +447296.612}
SPL {X  -162.820, Y  +465.727, Z    +0.000, E1   +25.676, E3 +447313.655}
SPL {X  -162.820, Y  +463.001, Z    +0.000, E1   +25.614, E3 +447325.771}
SPL {X  -162.820, Y  +459.882, Z    +0.000, E1   +25.674, E3 +447339.072}
SPL {X  -162.820, Y  +456.773, Z    +0.000, E1   +25.591, E3 +447353.018}
SPL {X  -162.820, Y  +454.429, Z    +0.000, E1   +25.642, E3 +447362.786}
SPL {X  -162.820, Y  +451.204, Z    +0.000, E1   +25.672, E3 +447376.812}
SPL {X  -162.820, Y  +447.822, Z    +0.000, E1   +25.664, E3 +447391.296}
SPL {X  -162.820, Y  +445.556, Z    +0.000, E1   +25.626, E3 +447401.427}
SPL {X  -162.820, Y  +442.508, Z    +0.000, E1   +25.657, E3 +447414.521}
SPL {X  -162.820, Y  +439.273, Z    +0.000, E1   +25.576, E3 +447429.159}
SPL {X  -162.820, Y  +436.773, Z    +0.000, E1   +25.602, E3 +447439.724}
SPL {X  -162.820, Y  +433.761, Z    +0.000, E1   +25.681, E3 +447452.402}
SPL {X  -162.820, Y  +430.942, Z    +0.000, E1   +25.597, E3 +447465.087}
SPL {X  -162.820, Y  +428.576, Z    +0.000, E1   +25.647, E3 +447475.025}
SPL {X  -162.820, Y  +426.525, Z    +0.000, E1   +25.610, E3 +447484.132}
SPL {X  -162.820, Y  +423.655, Z    +0.000, E1   +25.628, E3 +447496.692}
SPL {X  -162.820, Y  +419.407, Z    +0.000, E1   +25.665, E3 +447514.884}
SPL {X  -162.820, Y  +415.900, Z    +0.000, E1   +25.638, E3 +447530.154}
SPL {X  -162.820, Y  +413.088, Z    +0.000, E1   +25.644, E3 +447542.310}
SPL {X  -162.820, Y  +410.320, Z    +0.000, E1   +25.604, E3 +447554.629}
SPL {X  -162.820, Y  +407.487, Z    +0.000, E1   +25.617, E3 +447566.837}
SPL {X  -162.820, Y  +405.108, Z    +0.000, E1   +25.535, E3 +447577.804}
SPL {X  -162.820, Y  +401.373, Z    +0.000, E1   +25.736, E3 +447592.641}
SPL {X  -162.820, Y  +398.703, Z    +0.000, E1   +25.586, E3 +447605.138}
SPL {X  -162.820, Y  +395.582, Z    +0.000, E1   +25.684, E3 +447618.129}
SPL {X  -162.820, Y  +391.417, Z    +0.000, E1   +25.659, E3 +447636.467}
SPL {X  -162.820, Y  +387.939, Z    +0.000, E1   +25.627, E3 +447651.614}
SPL {X  -162.820, Y  +385.565, Z    +0.000, E1   +25.686, E3 +447661.403}
SPL {X  -162.820, Y  +383.458, Z    +0.000, E1   +25.657, E3 +447670.767}
SPL {X  -162.820, Y  +381.229, Z    +0.000, E1   +25.660, E3 +447680.442}
SPL {X  -162.797, Y  +377.786, Z    +0.000, E1   +25.638, E3 +447695.732}
SPL {X  -162.663, Y  +373.346, Z    +0.000, E1   +25.707, E3 +447714.471}
SPL {X  -162.487, Y  +370.088, Z    +0.000, E1   +25.525, E3 +447729.805}
SPL {X  -162.307, Y  +367.587, Z    +0.000, E1   +25.577, E3 +447740.224}
SPL {X  -162.041, Y  +364.588, Z    +0.000, E1   +25.591, E3 +447753.301}
SPL {X  -161.695, Y  +361.389, Z    +0.000, E1   +25.445, E3 +447768.187}
SPL {X  -161.190, Y  +357.520, Z    +0.000, E1   +25.774, E3 +447782.439}
SPL {X  -155.035, Y  +330.756, Z    +0.000, E1   +37.918, E3 +447792.940}
SPL {X  -153.918, Y  +327.401, Z    +0.000, E1   +34.677, E3 +447828.240}
ENDSPLINE

SPLINE
SPL {X  -159.701, Y  +348.785, Z    +0.000, E1   +24.361, E3 +447835.721}
SPL {X  -161.904, Y  +363.251, Z    +0.000, E1   +14.606, E3 +447865.516}
SPL {X  -162.745, Y  +375.561, Z    +0.000, E1    +7.538, E3 +447865.713}
SPL {X  -162.820, Y  +385.424, Z    +0.000, E1    +1.080, E3 +447866.607}
SPL {X  -162.820, Y  +389.940, Z    +0.000, E1    -2.281, E3 +447869.484}
SPL {X  -162.820, Y  +396.652, Z    +0.000, E1    -7.520, E3 +447869.062}
SPL {X  -162.820, Y  +406.605, Z    +0.000, E1   -16.760, E3 +447861.539}
SPL {X  -162.820, Y  +420.013, Z    +0.000, E1   -22.833, E3 +447889.660}
SPL {X  -162.820, Y  +442.075, Z    +0.000, E1   -31.090, E3 +447922.446}
ENDSPLINE

SPLINE
SPL {X  -162.820, Y  +436.680, Z    +0.000, E1   -26.151, E3 +447935.751}
ENDSPLINE

SPLINE
SPL {X  -162.820, Y  +438.487, Z    +0.000, E1   -25.409, E3 +447949.389}
SPL {X  -162.820, Y  +441.593, Z    +0.000, E1   -25.391, E3 +447962.998}
SPL {X  -162.820, Y  +444.317, Z    +0.000, E1   -25.492, E3 +447974.179}
SPL {X  -162.820, Y  +447.641, Z    +0.000, E1   -25.460, E3 +447989.114}
SPL {X  -162.820, Y  +451.939, Z    +0.000, E1   -25.468, E3 +448007.934}
SPL {X  -162.820, Y  +455.480, Z    +0.000, E1   -25.454, E3 +448023.345}
SPL {X  -162.820, Y  +458.079, Z    +0.000, E1   -25.369, E3 +448035.381}
SPL {X  -162.820, Y  +460.719, Z    +0.000, E1   -25.411, E3 +448046.639}
SPL {X  -162.820, Y  +463.419, Z    +0.000, E1   -25.510, E3 +448057.677}
SPL {X  -162.820, Y  +466.458, Z    +0.000, E1   -25.433, E3 +448071.732}
SPL {X  -162.820, Y  +470.010, Z    +0.000, E1   -25.445, E3 +448087.101}
SPL {X  -162.820, Y  +472.345, Z    +0.000, E1   -25.448, E3 +448097.187}
SPL {X  -162.820, Y  +475.191, Z    +0.000, E1   -25.489, E3 +448109.550}
SPL {X  -162.820, Y  +478.461, Z    +0.000, E1   -25.410, E3 +448124.319}
SPL {X  -162.820, Y  +480.780, Z    +0.000, E1   -25.447, E3 +448134.181}
SPL {X  -162.820, Y  +483.622, Z    +0.000, E1   -25.381, E3 +448147.223}
SPL {X  -162.820, Y  +487.570, Z    +0.000, E1   -25.482, E3 +448163.861}
SPL {X  -162.820, Y  +491.017, Z    +0.000, E1   -25.445, E3 +448179.075}
SPL {X  -162.820, Y  +493.705, Z    +0.000, E1   -25.443, E3 +448190.860}
SPL {X  -162.820, Y  +497.247, Z    +0.000, E1   -25.470, E3 +448206.322}
SPL {X  -162.820, Y  +501.343, Z    +0.000, E1   -25.435, E3 +448224.521}
SPL {X  -162.820, Y  +505.370, Z    +0.000, E1   -25.456, E3 +448241.984}
SPL {X  -162.820, Y  +509.412, Z    +0.000, E1   -25.458, E3 +448259.707}
SPL {X  -162.820, Y  +512.406, Z    +0.000, E1   -25.425, E3 +448272.863}
SPL {X  -162.820, Y  +515.039, Z    +0.000, E1   -25.452, E3 +448284.274}
SPL {X  -162.820, Y  +518.350, Z    +0.000, E1   -25.425, E3 +448299.023}
SPL {X  -162.820, Y  +521.486, Z    +0.000, E1   -25.382, E3 +448313.051}
SPL {X  -162.820, Y  +524.180, Z    +0.000, E1   -25.495, E3 +448323.923}
SPL {X  -162.820, Y  +527.020, Z    +0.000, E1   -25.477, E3 +448336.616}
SPL {X  -162.820, Y  +529.670, Z    +0.000, E1   -25.472, E3 +448348.074}
SPL {X  -162.820, Y  +532.006, Z    +0.000, E1   -25.455, E3 +448358.531}
SPL {X  -162.820, Y  +534.806, Z    +0.000, E1   -25.465, E3 +448370.647}
SPL {X  -162.820, Y  +537.226, Z    +0.000, E1   -25.378, E3 +448381.929}
SPL {X  -162.820, Y  +540.345, Z    +0.000, E1   -25.451, E3 +448395.110}
SPL {X  -162.820, Y  +543.279, Z    +0.000, E1   -25.419, E3 +448408.143}
SPL {X  -162.820, Y  +546.125, Z    +0.000, E1   -25.505, E3 +448419.937}
SPL {X  -162.820, Y  +549.578, Z    +0.000, E1   -25.462, E3 +448435.561}
SPL {X  -162.820, Y  +553.157, Z    +0.000, E1   -25.443, E3 +448451.225}
SPL {X  -162.820, Y  +556.150, Z    +0.000, E1   -25.445, E3 +448464.314}
SPL {X  -162.820, Y  +559.215, Z    +0.000, E1   -25.460, E3 +448477.616}
SPL {X  -162.820, Y  +562.125, Z    +0.000, E1   -25.434, E3 +448490.536}
SPL {X  -162.820, Y  +564.880, Z    +0.000, E1   -25.448, E3 +448502.490}
SPL {X  -162.820, Y  +568.326, Z    +0.000, E1   -25.470, E3 +448517.550}
SPL {X  -162.820, Y  +571.303, Z    +0.000, E1   -25.427, E3 +448530.723}
SPL {X  -162.820, Y  +574.067, Z    +0.000, E1   -25.459, E3 +448542.662}
SPL {X  -162.820, Y  +576.597, Z    +0.000, E1   -25.400, E3 +448554.133}
SPL {X  -162.820, Y  +578.977, Z    +0.000, E1   -25.460, E3 +448564.066}
SPL {X  -162.820, Y  +581.995, Z    +0.000, E1   -25.468, E3 +448577.424}
SPL {X  -162.820, Y  +585.512, Z    +0.000, E1   -25.448, E3 +448592.847}
SPL {X  -162.820, Y  +588.371, Z    +0.000, E1   -25.460, E3 +448605.233}
SPL {X  -162.820, Y  +591.246, Z    +0.000, E1   -25.415, E3 +448618.252}
SPL {X  -162.820, Y  +594.339, Z    +0.000, E1   -25.487, E3 +448631.155}
SPL {X  -162.820, Y  +596.868, Z    +0.000, E1   -25.461, E3 +448642.418}
SPL {X  -162.820, Y  +600.326, Z    +0.000, E1   -25.438, E3 +448657.939}
SPL {X  -162.820, Y  +604.526, Z    +0.000, E1   -25.502, E3 +448675.762}
SPL {X  -162.820, Y  +607.811, Z    +0.000, E1   -25.507, E3 +448689.977}
SPL {X  -162.820, Y  +610.517, Z    +0.000, E1   -25.412, E3 +448702.539}
SPL {X  -162.820, Y  +613.762, Z    +0.000, E1   -25.472, E3 +448716.346}
SPL {X  -162.820, Y  +616.216, Z    +0.000, E1   -25.419, E3 +448727.342}
SPL {X  -162.820, Y  +618.995, Z    +0.000, E1   -25.483, E3 +448739.191}
SPL {X  -162.820, Y  +622.118, Z    +0.000, E1   -25.492, E3 +448752.656}
SPL {X  -162.820, Y  +624.430, Z    +0.000, E1   -25.475, E3 +448762.877}
SPL {X  -162.820, Y  +626.570, Z    +0.000, E1   -25.441, E3 +448772.478}
SPL {X  -162.820, Y  +628.902, Z    +0.000, E1   -25.449, E3 +448782.658}
SPL {X  -162.820, Y  +631.177, Z    +0.000, E1   -25.467, E3 +448792.489}
SPL {X  -162.820, Y  +633.994, Z    +0.000, E1   -25.503, E3 +448804.536}
SPL {X  -162.820, Y  +636.469, Z    +0.000, E1   -25.465, E3 +448815.579}
SPL {X  -162.820, Y  +638.486, Z    +0.000, E1   -25.456, E3 +448824.497}
SPL {X  -162.820, Y  +640.803, Z    +0.000, E1   -25.462, E3 +448834.559}
SPL {X  -162.820, Y  +643.028, Z    +0.000, E1   -25.494, E3 +448844.068}
SPL {X  -162.820, Y  +645.694, Z    +0.000, E1   -25.540, E3 +448855.356}
SPL {X  -162.820, Y  +649.102, Z    +0.000, E1   -25.495, E3 +448870.784}
SPL {X  -162.820, Y  +652.810, Z    +0.000, E1   -25.497, E3 +448886.817}
SPL {X  -162.820, Y  +655.214, Z    +0.000, E1   -25.485, E3 +448897.320}
SPL {X  -162.820, Y  +657.616, Z    +0.000, E1   -25.511, E3 +448907.674}
SPL {X  -162.820, Y  +660.007, Z    +0.000, E1   -25.550, E3 +448917.736}
SPL {X  -162.820, Y  +662.980, Z    +0.000, E1   -25.505, E3 +448931.294}
SPL {X  -162.820, Y  +667.253, Z    +0.000, E1   -25.483, E3 +448950.171}
SPL {X  -162.820, Y  +671.102, Z    +0.000, E1   -25.514, E3 +448966.621}
SPL {X  -162.820, Y  +673.648, Z    +0.000, E1   -25.431, E3 +448978.288}
SPL {X  -162.796, Y  +676.319, Z    +0.000, E1   -25.526, E3 +448989.297}
SPL {X  -162.707, Y  +679.552, Z    +0.000, E1   -25.443, E3 +449004.172}
SPL {X  -162.545, Y  +682.952, Z    +0.000, E1   -25.510, E3 +449018.405}
SPL {X  -162.381, Y  +685.455, Z    +0.000, E1   -25.410, E3 +449030.092}
SPL {X  -162.102, Y  +688.774, Z    +0.000, E1   -25.417, E3 +449044.706}
SPL {X  -161.711, Y  +692.468, Z    +0.000, E1   -25.300, E3 +449061.678}
SPL {X  -161.141, Y  +696.825, Z    +0.000, E1   -26.170, E3 +449073.813}
SPL {X  -157.976, Y  +712.921, Z    +0.000, E1   -33.197, E3 +449084.353}
ENDSPLINE

SPLINE
SPL {X  -160.738, Y  +699.453, Z    +0.000, E1   -21.994, E3 +449121.980}
SPL {X  -161.689, Y  +692.657, Z    +0.000, E1   -15.656, E3 +449162.050}
SPL {X  -162.807, Y  +675.545, Z    +0.000, E1    -5.787, E3 +449157.550}
ENDSPLINE

SPLINE
SPL {X  -162.791, Y  +676.574, Z    +0.000, E1    -6.127, E3 +449170.652}
ENDSPLINE

SPLINE
SPL {X  -162.820, Y  +664.716, Z    +0.000, E1    +1.705, E3 +449159.527}
SPL {X  -162.820, Y  +658.484, Z    +0.000, E1    +6.336, E3 +449166.003}
SPL {X  -162.820, Y  +640.102, Z    +0.000, E1   +22.409, E3 +449160.742}
SPL {X  -162.820, Y  +633.503, Z    +0.000, E1   +21.975, E3 +449192.978}
SPL {X  -162.820, Y  +611.299, Z    +0.000, E1   +31.088, E3 +449221.091}
ENDSPLINE

SPLINE
SPL {X  -162.820, Y  +618.877, Z    +0.000, E1   +25.259, E3 +449232.585}
ENDSPLINE

SPLINE
SPL {X  -162.820, Y  +617.582, Z    +0.000, E1   +24.552, E3 +449243.962}
SPL {X  -162.820, Y  +614.716, Z    +0.000, E1   +24.535, E3 +449257.173}
SPL {X  -162.820, Y  +611.754, Z    +0.000, E1   +24.563, E3 +449270.461}
SPL {X  -162.820, Y  +608.970, Z    +0.000, E1   +24.542, E3 +449283.302}
SPL {X  -162.820, Y  +606.285, Z    +0.000, E1   +24.533, E3 +449295.637}
SPL {X  -162.820, Y  +603.509, Z    +0.000, E1   +24.546, E3 +449308.174}
SPL {X  -162.820, Y  +600.818, Z    +0.000, E1   +24.590, E3 +449320.097}
SPL {X  -162.820, Y  +598.053, Z    +0.000, E1   +24.547, E3 +449333.080}
SPL {X  -162.820, Y  +595.188, Z    +0.000, E1   +24.538, E3 +449346.169}
SPL {X  -162.820, Y  +592.738, Z    +0.000, E1   +24.551, E3 +449357.217}
SPL {X  -162.820, Y  +590.118, Z    +0.000, E1   +24.544, E3 +449369.276}
SPL {X  -162.820, Y  +587.204, Z    +0.000, E1   +24.592, E3 +449382.153}
SPL {X  -162.820, Y  +584.766, Z    +0.000, E1   +24.499, E3 +449393.986}
SPL {X  -162.820, Y  +581.896, Z    +0.000, E1   +24.528, E3 +449406.928}
SPL {X  -162.820, Y  +579.244, Z    +0.000, E1   +24.610, E3 +449418.272}
SPL {X  -162.820, Y  +576.848, Z    +0.000, E1   +24.543, E3 +449429.814}
SPL {X  -162.820, Y  +573.694, Z    +0.000, E1   +24.535, E3 +449444.283}
SPL {X  -162.820, Y  +571.322, Z    +0.000, E1   +24.492, E3 +449455.317}
SPL {X  -162.820, Y  +568.309, Z    +0.000, E1   +24.589, E3 +449468.542}
SPL {X  -162.820, Y  +564.977, Z    +0.000, E1   +24.571, E3 +449483.715}
SPL {X  -162.820, Y  +562.356, Z    +0.000, E1   +24.575, E3 +449495.613}
SPL {X  -162.820, Y  +560.119, Z    +0.000, E1   +24.506, E3 +449506.302}
SPL {X  -162.820, Y  +558.093, Z    +0.000, E1   +24.537, E3 +449515.320}
SPL {X  -162.820, Y  +555.584, Z    +0.000, E1   +24.559, E3 +449526.632}
SPL {X  -162.820, Y  +552.169, Z    +0.000, E1   +24.581, E3 +449542.201}
SPL {X  -162.820, Y  +548.172, Z    +0.000, E1   +24.564, E3 +449560.549}
SPL {X  -162.820, Y  +544.025, Z    +0.000, E1   +24.611, E3 +449579.103}
SPL {X  -162.820, Y  +540.573, Z    +0.000, E1   +24.503, E3 +449595.558}
SPL {X  -162.820, Y  +538.106, Z    +0.000, E1   +24.553, E3 +449606.311}
SPL {X  -162.820, Y  +536.451, Z    +0.000, E1   +24.519, E3 +449614.130}
SPL {X  -162.820, Y  +534.025, Z    +0.000, E1   +24.589, E3 +449624.730}
SPL {X  -162.820, Y  +531.527, Z    +0.000, E1   +24.582, E3 +449636.115}
SPL {X  -162.820, Y  +529.165, Z    +0.000, E1   +24.521, E3 +449647.364}
SPL {X  -162.820, Y  +525.802, Z    +0.000, E1   +24.585, E3 +449662.384}
SPL {X  -162.820, Y  +521.731, Z    +0.000, E1   +24.542, E3 +449681.320}
SPL {X  -162.820, Y  +518.185, Z    +0.000, E1   +24.561, E3 +449697.192}
SPL {X  -162.820, Y  +508.728, Z    +0.000, E1   +28.484, E3 +449707.732}
SPL {X  -162.820, Y  +500.664, Z    +0.000, E1   +31.476, E3 +449716.396}
SPL {X  -162.820, Y  +499.290, Z    +0.000, E1   +30.657, E3 +449726.678}
SPL {X  -162.820, Y  +497.700, Z    +0.000, E1   +29.785, E3 +449738.293}
SPL {X  -162.820, Y  +495.915, Z    +0.000, E1   +28.861, E3 +449751.385}
SPL {X  -162.820, Y  +494.678, Z    +0.000, E1   +27.647, E3 +449764.731}
SPL {X  -162.820, Y  +493.757, Z    +0.000, E1   +26.462, E3 +449777.091}
SPL {X  -162.820, Y  +491.420, Z    +0.000, E1   +25.780, E3 +449792.353}
SPL {X  -162.820, Y  +487.351, Z    +0.000, E1   +25.663, E3 +449810.869}
SPL {X  -162.820, Y  +484.247, Z    +0.000, E1   +25.651, E3 +449824.195}
SPL {X  -162.820, Y  +482.092, Z    +0.000, E1   +25.593, E3 +449834.022}
SPL {X  -162.820, Y  +479.578, Z    +0.000, E1   +25.634, E3 +449844.665}
SPL {X  -162.820, Y  +477.137, Z    +0.000, E1   +25.632, E3 +449855.244}
SPL {X  -162.820, Y  +473.770, Z    +0.000, E1   +25.664, E3 +449869.790}
SPL {X  -162.820, Y  +469.694, Z    +0.000, E1   +25.657, E3 +449887.521}
SPL {X  -162.820, Y  +465.727, Z    +0.000, E1   +25.676, E3 +449904.564}
SPL {X  -162.820, Y  +463.001, Z    +0.000, E1   +25.614, E3 +449916.680}
SPL {X  -162.820, Y  +459.882, Z    +0.000, E1   +25.674, E3 +449929.981}
SPL {X  -162.820, Y  +456.773, Z    +0.000, E1   +25.591, E3 +449943.927}
SPL {X  -162.820, Y  +454.429, Z    +0.000, E1   +25.642, E3 +449953.695}
SPL {X  -162.820, Y  +451.204, Z    +0.000, E1   +25.672, E3 +449967.722}
SPL {X  -162.820, Y  +447.822, Z    +0.000, E1   +25.664, E3 +449982.205}
SPL {X  -162.820, Y  +445.556, Z    +0.000, E1   +25.626, E3 +449992.336}
SPL {X  -162.820, Y  +443.328, Z    +0.000, E1   +25.642, E3 +450001.850}
SPL {X  -162.820, Y  +440.857, Z    +0.000, E1   +25.614, E3 +450012.884}
SPL {X  -162.820, Y  +437.636, Z    +0.000, E1   +25.597, E3 +450027.048}
SPL {X  -162.820, Y  +434.768, Z    +0.000, E1   +25.655, E3 +450038.950}
SPL {X  -162.820, Y  +431.823, Z    +0.000, E1   +25.651, E3 +450051.949}
SPL {X  -162.820, Y  +427.740, Z    +0.000, E1   +25.667, E3 +450069.577}
SPL {X  -162.820, Y  +423.655, Z    +0.000, E1   +25.628, E3 +450087.601}
SPL {X  -162.820, Y  +419.407, Z    +0.000, E1   +25.665, E3 +450105.794}
SPL {X  -162.820, Y  +415.900, Z    +0.000, E1   +25.638, E3 +450121.063}
SPL {X  -162.820, Y  +413.088, Z    +0.000, E1   +25.644, E3 +450133.219}
SPL {X  -162.820, Y  +410.320, Z    +0.000, E1   +25.604, E3 +450145.538}
SPL {X  -162.820, Y  +407.487, Z    +0.000, E1   +25.617, E3 +450157.746}
SPL {X  -162.820, Y  +405.108, Z    +0.000, E1   +25.535, E3 +450168.713}
SPL {X  -162.820, Y  +401.373, Z    +0.000, E1   +25.736, E3 +450183.550}
SPL {X  -162.820, Y  +397.357, Z    +0.000, E1   +25.652, E3 +450201.620}
SPL {X  -162.820, Y  +393.659, Z    +0.000, E1   +25.666, E3 +450217.420}
SPL {X  -162.820, Y  +390.679, Z    +0.000, E1   +25.624, E3 +450230.664}
SPL {X  -162.820, Y  +387.939, Z    +0.000, E1   +25.627, E3 +450242.523}
SPL {X  -162.820, Y  +384.398, Z    +0.000, E1   +25.707, E3 +450257.421}
SPL {X  -162.820, Y  +380.448, Z    +0.000, E1   +25.674, E3 +450274.784}
SPL {X  -162.785, Y  +377.106, Z    +0.000, E1   +25.598, E3 +450289.729}
SPL {X  -162.709, Y  +374.484, Z    +0.000, E1   +25.711, E3 +450300.180}
SPL {X  -162.623, Y  +372.485, Z    +0.000, E1   +25.631, E3 +450309.460}
SPL {X  -162.487, Y  +370.088, Z    +0.000, E1   +25.525, E3 +450320.714}
SPL {X  -162.243, Y  +366.801, Z    +0.000, E1   +25.618, E3 +450334.355}
SPL {X  -161.977, Y  +363.953, Z    +0.000, E1   +25.528, E3 +450347.281}
SPL {X  -161.695, Y  +361.389, Z    +0.000, E1   +25.445, E3 +450359.096}
SPL {X  -161.364, Y  +358.774, Z    +0.000, E1   +25.454, E3 +450370.297}
SPL {X  -160.939, Y  +355.820, Z    +0.000, E1   +26.179, E3 +450377.515}
SPL {X  -155.035, Y  +330.756, Z    +0.000, E1   +37.918, E3 +450383.849}
SPL {X  -153.918, Y  +327.401, Z    +0.000, E1   +34.677, E3 +450419.150}
ENDSPLINE

SPLINE
SPL {X  -159.701, Y  +348.785, Z    +0.000, E1   +24.361, E3 +450426.630}
SPL {X  -162.442, Y  +369.407, Z    +0.000, E1   +11.234, E3 +450456.265}
SPL {X  -162.820, Y  +384.333, Z    +0.000, E1    +1.902, E3 +450457.471}
SPL {X  -162.820, Y  +389.940, Z    +0.000, E1    -2.281, E3 +450460.393}
SPL {X  -162.820, Y  +396.652, Z    +0.000, E1    -7.520, E3 +450459.971}
SPL {X  -162.820, Y  +406.605, Z    +0.000, E1   -16.760, E3 +450452.448}
SPL {X  -162.820, Y  +418.675, Z    +0.000, E1   -22.201, E3 +450478.697}
SPL {X  -162.820, Y  +425.113, Z    +0.000, E1   -25.243, E3 +450487.633}
SPL {X  -162.820, Y  +441.937, Z    +0.000, E1   -31.578, E3 +450509.711}
ENDSPLINE

SPLINE
SPL {X  -162.820, Y  +437.771, Z    +0.000, E1   -26.555, E3 +450528.812}
ENDSPLINE

SPLINE
SPL {X  -162.820, Y  +439.120, Z    +0.000, E1   -25.352, E3 +450543.355}
SPL {X  -162.820, Y  +441.593, Z    +0.000, E1   -25.391, E3 +450553.907}
SPL {X  -162.820, Y  +444.317, Z    +0.000, E1   -25.492, E3 +450565.088}
SPL {X  -162.820, Y  +446.544, Z    +0.000, E1   -25.427, E3 +450575.258}
SPL {X  -162.820, Y  +448.500, Z    +0.000, E1   -25.425, E3 +450583.859}
SPL {X  -162.820, Y  +451.056, Z    +0.000, E1   -25.443, E3 +450594.966}
SPL {X  -162.820, Y  +454.662, Z    +0.000, E1   -25.474, E3 +450610.711}
SPL {X  -162.820, Y  +458.079, Z    +0.000, E1   -25.369, E3 +450626.290}
SPL {X  -162.820, Y  +460.719, Z    +0.000, E1   -25.411, E3 +450637.548}
SPL {X  -162.820, Y  +463.419, Z    +0.000, E1   -25.510, E3 +450648.586}
SPL {X  -162.820, Y  +465.376, Z    +0.000, E1   -25.372, E3 +450658.174}
SPL {X  -162.820, Y  +467.440, Z    +0.000, E1   -25.427, E3 +450666.805}
SPL {X  -162.820, Y  +470.010, Z    +0.000, E1   -25.445, E3 +450678.010}
SPL {X  -162.820, Y  +473.445, Z    +0.000, E1   -25.493, E3 +450692.734}
SPL {X  -162.820, Y  +476.157, Z    +0.000, E1   -25.426, E3 +450704.948}
SPL {X  -162.820, Y  +478.461, Z    +0.000, E1   -25.410, E3 +450715.228}
SPL {X  -162.820, Y  +481.644, Z    +0.000, E1   -25.433, E3 +450729.175}
SPL {X  -162.820, Y  +486.042, Z    +0.000, E1   -25.483, E3 +450748.094}
SPL {X  -162.820, Y  +490.287, Z    +0.000, E1   -25.463, E3 +450766.812}
SPL {X  -162.820, Y  +494.454, Z    +0.000, E1   -25.465, E3 +450785.044}
SPL {X  -162.820, Y  +498.644, Z    +0.000, E1   -25.463, E3 +450803.420}
SPL {X  -162.820, Y  +502.845, Z    +0.000, E1   -25.458, E3 +450821.853}
SPL {X  -162.820, Y  +506.050, Z    +0.000, E1   -25.420, E3 +450835.993}
SPL {X  -162.820, Y  +508.346, Z    +0.000, E1   -25.444, E3 +450845.841}
SPL {X  -162.820, Y  +510.377, Z    +0.000, E1   -25.398, E3 +450855.087}
SPL {X  -162.820, Y  +513.176, Z    +0.000, E1   -25.443, E3 +450867.131}
SPL {X  -162.820, Y  +516.690, Z    +0.000, E1   -25.465, E3 +450882.342}
SPL {X  -162.820, Y  +519.134, Z    +0.000, E1   -25.366, E3 +450893.664}
SPL {X  -162.820, Y  +521.486, Z    +0.000, E1   -25.382, E3 +450903.960}
SPL {X  -162.820, Y  +524.180, Z    +0.000, E1   -25.495, E3 +450914.832}
SPL {X  -162.820, Y  +527.020, Z    +0.000, E1   -25.477, E3 +450927.525}
SPL {X  -162.820, Y  +529.670, Z    +0.000, E1   -25.472, E3 +450938.983}
SPL {X  -162.820, Y  +532.006, Z    +0.000, E1   -25.455, E3 +450949.440}
SPL {X  -162.820, Y  +534.806, Z    +0.000, E1   -25.465, E3 +450961.556}
SPL {X  -162.820, Y  +537.226, Z    +0.000, E1   -25.378, E3 +450972.838}
SPL {X  -162.820, Y  +540.345, Z    +0.000, E1   -25.451, E3 +450986.019}
SPL {X  -162.820, Y  +543.279, Z    +0.000, E1   -25.419, E3 +450999.052}
SPL {X  -162.820, Y  +546.125, Z    +0.000, E1   -25.505, E3 +451010.846}
SPL {X  -162.820, Y  +549.578, Z    +0.000, E1   -25.462, E3 +451026.470}
SPL {X  -162.820, Y  +553.157, Z    +0.000, E1   -25.443, E3 +451042.134}
SPL {X  -162.820, Y  +556.150, Z    +0.000, E1   -25.445, E3 +451055.223}
SPL {X  -162.820, Y  +559.215, Z    +0.000, E1   -25.460, E3 +451068.525}
SPL {X  -162.820, Y  +562.125, Z    +0.000, E1   -25.434, E3 +451081.445}
SPL {X  -162.820, Y  +564.880, Z    +0.000, E1   -25.448, E3 +451093.400}
SPL {X  -162.820, Y  +568.326, Z    +0.000, E1   -25.470, E3 +451108.459}
SPL {X  -162.820, Y  +571.303, Z    +0.000, E1   -25.427, E3 +451121.632}
SPL {X  -162.820, Y  +574.067, Z    +0.000, E1   -25.459, E3 +451133.571}
SPL {X  -162.820, Y  +576.597, Z    +0.000, E1   -25.400, E3 +451145.042}
SPL {X  -162.820, Y  +578.977, Z    +0.000, E1   -25.460, E3 +451154.975}
SPL {X  -162.820, Y  +581.995, Z    +0.000, E1   -25.468, E3 +451168.333}
SPL {X  -162.820, Y  +585.512, Z    +0.000, E1   -25.448, E3 +451183.756}
SPL {X  -162.820, Y  +588.371, Z    +0.000, E1   -25.460, E3 +451196.142}
SPL {X  -162.820, Y  +591.246, Z    +0.000, E1   -25.415, E3 +451209.161}
SPL {X  -162.820, Y  +594.339, Z    +0.000, E1   -25.487, E3 +451222.064}
SPL {X  -162.820, Y  +596.868, Z    +0.000, E1   -25.461, E3 +451233.327}
SPL {X  -162.820, Y  +599.135, Z    +0.000, E1   -25.398, E3 +451243.696}
SPL {X  -162.820, Y  +601.296, Z    +0.000, E1   -25.399, E3 +451253.178}
SPL {X  -162.820, Y  +603.808, Z    +0.000, E1   -25.554, E3 +451262.966}
SPL {X  -162.820, Y  +607.007, Z    +0.000, E1   -25.491, E3 +451277.657}
SPL {X  -162.820, Y  +611.438, Z    +0.000, E1   -25.467, E3 +451297.247}
SPL {X  -162.820, Y  +615.388, Z    +0.000, E1   -25.455, E3 +451314.505}
SPL {X  -162.820, Y  +618.103, Z    +0.000, E1   -25.456, E3 +451326.253}
SPL {X  -162.820, Y  +621.264, Z    +0.000, E1   -25.514, E3 +451339.856}
SPL {X  -162.820, Y  +624.430, Z    +0.000, E1   -25.475, E3 +451353.787}
SPL {X  -162.820, Y  +626.570, Z    +0.000, E1   -25.441, E3 +451363.387}
SPL {X  -162.820, Y  +628.902, Z    +0.000, E1   -25.449, E3 +451373.567}
SPL {X  -162.820, Y  +631.177, Z    +0.000, E1   -25.467, E3 +451383.399}
SPL {X  -162.820, Y  +633.994, Z    +0.000, E1   -25.503, E3 +451395.445}
SPL {X  -162.820, Y  +636.469, Z    +0.000, E1   -25.465, E3 +451406.488}
SPL {X  -162.820, Y  +638.486, Z    +0.000, E1   -25.456, E3 +451415.406}
SPL {X  -162.820, Y  +640.803, Z    +0.000, E1   -25.462, E3 +451425.468}
SPL {X  -162.820, Y  +643.028, Z    +0.000, E1   -25.494, E3 +451434.977}
SPL {X  -162.820, Y  +645.694, Z    +0.000, E1   -25.540, E3 +451446.265}
SPL {X  -162.820, Y  +649.102, Z    +0.000, E1   -25.495, E3 +451461.693}
SPL {X  -162.820, Y  +652.810, Z    +0.000, E1   -25.497, E3 +451477.726}
SPL {X  -162.820, Y  +655.214, Z    +0.000, E1   -25.485, E3 +451488.229}
SPL {X  -162.820, Y  +657.616, Z    +0.000, E1   -25.511, E3 +451498.583}
SPL {X  -162.820, Y  +660.007, Z    +0.000, E1   -25.550, E3 +451508.645}
SPL {X  -162.820, Y  +662.980, Z    +0.000, E1   -25.505, E3 +451522.203}
SPL {X  -162.820, Y  +666.096, Z    +0.000, E1   -25.408, E3 +451536.374}
SPL {X  -162.820, Y  +668.238, Z    +0.000, E1   -25.482, E3 +451545.191}
SPL {X  -162.820, Y  +671.102, Z    +0.000, E1   -25.514, E3 +451557.530}
SPL {X  -162.820, Y  +673.648, Z    +0.000, E1   -25.431, E3 +451569.197}
SPL {X  -162.796, Y  +676.319, Z    +0.000, E1   -25.526, E3 +451580.206}
SPL {X  -162.707, Y  +679.552, Z    +0.000, E1   -25.443, E3 +451595.081}
SPL {X  -162.545, Y  +682.952, Z    +0.000, E1   -25.510, E3 +451609.314}
SPL {X  -162.381, Y  +685.455, Z    +0.000, E1   -25.410, E3 +451621.001}
SPL {X  -162.102, Y  +688.774, Z    +0.000, E1   -25.417, E3 +451635.615}
SPL {X  -161.711, Y  +692.468, Z    +0.000, E1   -25.300, E3 +451652.588}
SPL {X  -160.732, Y  +699.494, Z    +0.000, E1   -27.462, E3 +451666.060}
SPL {X  -157.189, Y  +715.948, Z    +0.000, E1   -34.218, E3 +451678.218}
ENDSPLINE

SPLINE
SPL {X  -160.780, Y  +699.193, Z    +0.000, E1   -22.069, E3 +451710.130}
ENDSPLINE

SPLINE
SPL {X  -160.671, Y  +699.864, Z    +0.000, E1   -21.788, E3 +451717.561}
ENDSPLINE

SPLINE
SPL {X  -160.945, Y  +698.140, Z    +0.000, E1   -18.412, E3 +451755.129}
SPL {X  -162.497, Y  +683.755, Z    +0.000, E1   -10.754, E3 +451749.273}
SPL {X  -162.819, Y  +673.996, Z    +0.000, E1    -4.745, E3 +451748.874}
ENDSPLINE

SPLINE
SPL {X  -162.791, Y  +676.574, Z    +0.000, E1    -6.127, E3 +451761.562}
ENDSPLINE

SPLINE
SPL {X  -162.820, Y  +666.063, Z    +0.000, E1    +0.780, E3 +451749.655}
SPL {X  -162.820, Y  +659.251, Z    +0.000, E1    +5.716, E3 +451755.871}
SPL {X  -162.820, Y  +640.102, Z    +0.000, E1   +22.409, E3 +451751.651}
SPL {X  -162.820, Y  +633.503, Z    +0.000, E1   +21.975, E3 +451783.887}
SPL {X  -162.820, Y  +611.299, Z    +0.000, E1   +31.088, E3 +451812.000}
ENDSPLINE

SPLINE
SPL {X  -162.820, Y  +618.877, Z    +0.000, E1   +25.259, E3 +451823.494}
ENDSPLINE

